(* CODESYS project SIMAI_1.0.0.project

Project tree, tasks and I/O mapping:
  Device : HY-TTC 540, TTControl, order no. n/a, version 1.7.1.0
    application Application
      libraries: Standard, * (System); CAA Can Low Level Extern, * (CAA Technical Workgroup); Util, * (System); SysTypes2 Interfaces, * (System); SysTarget, 3.5.5.0 (System); VisuDialogs, * (System); CAA Memory, 3.5.12.0 (CAA Technical Workgroup); Network, 3.5.7.0 (3S - Smart Software Solutions GmbH); CmpIecTask, * (System); CmpErrors, 3.3.1.40 (System); lib500, 1.7.1.0 (TTControl); lib500_types, 1.7.1.0 (TTControl); lib500_syscom, 1.7.1.0 (TTControl)
      task _NotificationCallback (externalevent, external event NotificationCallback, priority 0) calls _NotificationCB_PRG
      task _ErrorCallback (externalevent, external event ErrorCallback, priority 1) calls _ErrorCB_PRG
      task CommunicationTask (cyclic, interval t#10ms, priority 31, watchdog t#200ms x 1) calls manageGrCommAndEEPROM, CanComunication
      task MainTask (cyclic, interval t#10ms, priority 2, watchdog t#200ms x 1) calls MAIN
      Variable lists/
        global variables GVL
        global variables IO
        global variables fieldbus
        global variables par
        global variables CONST
        global variables ERR
        global variables ui
        global variables CanBusVariables
        global variables EtsdnVar
        global variables EtsOneVar
        global variables system
        global variables RxFlasher
      Program logic/
        program _ErrorCB_PRG [ST]
        program _NotificationCB_PRG [ST]
        Tasks/
          program MAIN [ST]: mainLoop, postrun, shutdown, checkParameters, setupCanbus
          program manageGrCommAndEEPROM [ST]: setVariablesToGrComm, initializeGrCommVariables, initializeEepromStructures
          program CanComunication [ST]: sendVariablesDisplay, receiveVariables, initialize, SendVariablesFromEtsdn, SendVariablesFromEtsOne
        function initializeCanbus [ST]
        program mngCanbusStatus [ST]: checkCanBusStatus
        program UI_PRG [ST]
        TypeApplication/
          program ETSDN_Test_PRG [ST]: endTest, setTestDuration, resetVariablesAndStartTest, mngFailTimer, isRLCurrentFresh
      STRUCTURES/
        data type EEPROM_FLAG
        data type CanHandleStatus
        data type FsmEnum
      Modules/
        IOs/
          Functions/
            program io_module [ST]: instantiateDI, instantiatePWM, instantiatePower, instantiateVOUT, instantiateADC, getInputs, instantiatePWD, initializeIO, instantiateDO, instantiateDIO, instantiatePVG, setOutputs, mngErrors
          Types/
            data type pinPWM
            program initializeIO [ST]: instantiateAnalogInputs, instantiatePVGOutputs, instantiateDigitalOutputs, instantiateVoltageOutputs, instantiatePWDInputs, instantiatePowerStages, instantiatePWMOutputs, instantiateDigitalInputs
            data type type_powerStages
            data type pinADC
            data type type_digitalInputs
            data type pinPVG
            data type type_pwmOutputs
            data type pinPWD
            data type type_voltageOutputs
            data type pinDIO
            data type pwdReadMode
            data type type_digitalOutputs
            data type type_analogInputs
            data type type_pwdInputs
            data type type_pvgOutputs
            data type pin
            data type pinPower
            data type pinVOUT
          global variables sysIO
        COMM/
          Functions/
            program mngCommCan [ST]: mngInit, catchMessages, mngMessage, mngResponse, getsetVarCallback, applyToRamCallback, readAllFromEEPROMCallback, writeToEEPROMCallback, applyToRAM, isVariableValid, initializeVariable
          Types/
            data type grCommVar
            data type grCommAccessRight
            data type grCommVariableStatus
            data type grCommMessageType
            data type grCommEEPROMStatus
          Variable lists/
            global variables grComm
        Canbus/
          Safety interface/
            Tasks/
              program CAN_PRG_SAFE [ST]: exchangeVariables
              program CAN_PRG_UNSAFE [ST]
            Functions/
              program safeSendMessage [ST]
              program safetyCanbusInterface [ST]
              program safeRegisterReceiveMask [ST]
          Variable lists/
            global variables canGVL
            global variables canEVL
          Types/
            data type can
            data type canMessage
            data type canReceiveMask
            data type canBus
          Functions/
            function readMessage [ST]
            program checkReceiveMaskInitialization [ST]
            program registerReceiveMask [ST]
            program sendMessage [ST]
            program initializeCanHandle [ST]
            program checkBusState [ST]
        EEPROM/
          Functions/
            program mngEEPROM [ST]: initEEPROM, mngStep, initializeEepromEntry
          Types/
            Parameters/
              data type HWFW_INFO_TIP
            data type eepromEntry
          Variable lists/
            global variables EEPROM
        Utils/
          program Utils [ST]: decrementUINT, bytesToUInt16, toggle, isNaN, updateValueFiltered, bytesToInt16, decrementUDINT, boolToPWMDutyCycle, linearize, bytesToUReal16, bytesToUDInt32, incrementUINT, getCurrentTaskCycleTime, decrementUINTTimer
        J1939/
          program J1939_PRG [ST]: initReceiveMasks, receiveMessage, parseMessage, sendPGNRequests, mngEngineStatus, redirectToDisplay
          global variables J1939
      visualisation Visualization
    CANs : CANs, TTControl, order no. n/a, version 1.7.1.0
      CAN2 : CAN2, TTControl, order no. n/a, version 1.7.1.0
      CAN3 : CAN3, TTControl, order no. n/a, version 1.7.1.0
      CAN0 : CAN0, TTControl, order no. n/a, version 1.7.1.0
      CAN1 : CAN1, TTControl, order no. n/a, version 1.7.1.0
    System_1 : System, TTControl, order no. n/a, version 1.7.1.0
        unmapped channels: mode, error, mode, error, mode, error, mode, error, mode, error, mode, error, shutdown, error, enable_error_group_0, enable_error_group_1, diag_status, safe_state, error, driver_init_error, UBAT, Terminal_15, WakeUp, Temperature, SSW0, SSW1, SSUP0, SSUP1, SSUP2, status, write, boot_error, trigger_error, Powerstage, SSW0, SSW1, SSUP0, SSUP1, SSUP2, Terminal_15,
          WakeUp, ExtShutOff0, ExtShutOff1
      Timer_Inputs : TIN, TTControl, order no. n/a, version 1.7.1.0
        Pin 147
          <Vuoto>
        Pin 122
          <Vuoto>
        Pin 148
          <Vuoto>
        Pin 146
          <Vuoto>
        Pin 124
          <Vuoto>
        Pin 123
          <Vuoto>
      Analog_Inputs_2Mode_10V : AIN_2Mode_10V, TTControl, order no. n/a, version 1.7.1.0
        Pin 134
          <Vuoto>
        Pin 109
          <Vuoto>
        Pin 132
          <Vuoto>
        Pin 131
          <Vuoto>
        Pin 107
          <Vuoto>
        Pin 110
          <Vuoto>
        Pin 108
          <Vuoto>
        Pin 133
          <Vuoto>
      Analog_Inputs_3Mode : AIN_3Mode, TTControl, order no. n/a, version 1.7.1.0
        Pin 129
          <Vuoto>
        Pin 104
          <Vuoto>
        Pin 130
          <Vuoto>
        Pin 105
          <Vuoto>
        Pin 103
          <Vuoto>
        Pin 127
          <Vuoto>
        Pin 106
          <Vuoto>
        Pin 128
          <Vuoto>
      Digital_Outputs_LS : LSDOUT, TTControl, order no. n/a, version 1.7.1.0
        Pin 239
          <Vuoto>
        Pin 251
          <Vuoto>
        Pin 240
          <Vuoto>
        Pin 252
          <Vuoto>
        Pin 254
          <Vuoto>
        Pin 238
          <Vuoto>
        Pin 253
          <Vuoto>
        Pin 241
          <Vuoto>
      Timer_Inputs_Cur : TIN_Cur, TTControl, order no. n/a, version 1.7.1.0
        Pin 140
          <Vuoto>
        Pin 117
          <Vuoto>
        Pin 116
          <Vuoto>
        Pin 139
          <Vuoto>
        Pin 115
          <Vuoto>
        Pin 141
          <Vuoto>
      Analog_Inputs_2Mode_32V : AIN_2Mode_32V, TTControl, order no. n/a, version 1.7.1.0
        Pin 113
          <Vuoto>
        Pin 137
          <Vuoto>
        Pin 136
          <Vuoto>
        Pin 112
          <Vuoto>
        Pin 138
          <Vuoto>
        Pin 114
          <Vuoto>
        Pin 111
          <Vuoto>
        Pin 135
          <Vuoto>
      PWM_Outputs : PWM, TTControl, order no. n/a, version 1.7.1.0
        Safety_switch_0 : PWM_SSW0, TTControl, order no. n/a, version 1.7.1.0
          Pin 165
            <Vuoto>
          Pin 195
            <Vuoto>
          Pin 162
            <Vuoto>
          Pin 171
            <Vuoto>
          Pin 168
            <Vuoto>
          Pin 186
            <Vuoto>
          Pin 183
            <Vuoto>
          Pin 177
            <Vuoto>
          Pin 180
            <Vuoto>
          Pin 159
            <Vuoto>
          Pin 153
            <Vuoto>
          Pin 189
            <Vuoto>
          Pin 156
            <Vuoto>
          Pin 192
            <Vuoto>
        Safety_switch_1 : PWM_SSW1, TTControl, order no. n/a, version 1.7.1.0
          Pin 157
            <Vuoto>
          Pin 187
            <Vuoto>
          Pin 154
            <Vuoto>
          Pin 160
            <Vuoto>
          Pin 178
            <Vuoto>
          Pin 169
            <Vuoto>
          Pin 166
            <Vuoto>
          Pin 163
            <Vuoto>
          Pin 184
            <Vuoto>
          Pin 181
            <Vuoto>
          Pin 190
            <Vuoto>
          Pin 172
            <Vuoto>
          Pin 193
            <Vuoto>
          Pin 196
            <Vuoto>
      Digital_Outputs_HS : HSDOUT, TTControl, order no. n/a, version 1.7.1.0
        Pin 176
          <Vuoto>
        Pin 149
          <Vuoto>
        Pin 158
          <Vuoto>
        Pin 173
          <Vuoto>
        Pin 152
          <Vuoto>
        Pin 155
          <Vuoto>
        Pin 182
          <Vuoto>
        Pin 179
          <Vuoto>
      Analog_Inputs : AIN, TTControl, order no. n/a, version 1.7.1.0
        Pin 161
          <Vuoto>
        Pin 185
          <Vuoto>
        Pin 188
          <Vuoto>
        Pin 164
          <Vuoto>
        Pin 191
          <Vuoto>
        Pin 167
          <Vuoto>
        Pin 194
          <Vuoto>
        Pin 170
          <Vuoto>
      Digital_Inputs : DIN, TTControl, order no. n/a, version 1.7.1.0
        Pin 101
          <Vuoto>
        Pin 125
          <Vuoto>
        Pin 150
          <Vuoto>
        Pin 174
          <Vuoto>
        Pin 102
          <Vuoto>
        Pin 126
          <Vuoto>
        Pin 151
          <Vuoto>
        Pin 175
          <Vuoto>
  text list GlobalTextList
*)

// Device/Application/STRUCTURES/EEPROM_FLAG
TYPE EEPROM_FLAG : //verificata
STRUCT
	READ: BOOL:= FALSE;
	CHANGED: BOOL:= FALSE;
	WRITE: BOOL:= FALSE;
END_STRUCT
END_TYPE

// Device/Application/Modules/COMM/Types/grCommVar
TYPE grCommVar :
	STRUCT;
		accessRights: grCommAccessRight;
		status: grCommVariableStatus;
		
		pointerToSystemVar: POINTER TO UINT;
		uiLowerValidValue: UINT;
		uiHigherValidValue: UINT;
		uiDefaultValue: UINT;
		
		uiValue: UINT;
	END_STRUCT
END_TYPE

// Device/Application/Modules/COMM/Types/grCommAccessRight
{attribute 'qualified_only'}
{attribute 'strict'}
TYPE grCommAccessRight :
(
	NoAccess := 0,
	ReadOnly := 1,
	ReadWrite := 2
);
END_TYPE

// Device/Application/Modules/COMM/Types/grCommVariableStatus
{attribute 'qualified_only'}
{attribute 'strict'}
TYPE grCommVariableStatus :
(
	Uninitialized:= 0,
	Pristine:= 1,
	ModifiedByRemote:= 2,
	Error:= 3
);
END_TYPE

// Device/Application/Modules/COMM/Types/grCommMessageType
{attribute 'qualified_only'}
{attribute 'strict'}
TYPE grCommMessageType :
(
	ExitCode:= 0,				// Esito di un comando
	
	GetVariable:= 1,			// Get valore di una variabile
	SetVariable:= 2,			// Set valore di una variabile
	HeartRateRequest:= 3,		// Richiesta di heart rate (broadcast)
	LoadFromEEPROM:= 4,			// Leggi parametri da EEPROM
	WriteToEEPROM:= 5,			// Scrivi parametri in RAM sulla EEPROM (rispettando il flag EDIT)
	WriteAllToEEPROM:= 6,		// Scrivi parametri in RAM sulla EEPROM (ignorando il flag EDIT)
	ApplyVariables:= 7,			// Imposta i parametri inviati sulla RAM
	
	ErrorCode:= 255		// Errore
);
END_TYPE

// Device/Application/Modules/IOs/Types/pinPWM
TYPE pinPWM EXTENDS pin :
	STRUCT
		stErrorGetCut: lib500_types.IO_ERRORTYPE;
		wFrequency: WORD:= 100;
		bPolarity: BOOL:= TRUE;
		bDiagMargin: BOOL:= FALSE;
		wFeedbackHighTime: WORD;
		wPeriodFeedback: WORD;
		wCurrent: WORD;
		bCurrentFresh: BOOL;
		wDuty: WORD;
	END_STRUCT
END_TYPE

// Device/Application/Modules/IOs/Types/type_powerStages
TYPE type_powerStages :
STRUCT	
	safetySwitch0: pinPower;	
	safetySwitch1: pinPower;	
	safetySwitch2: pinPower;
	powerStage: pinPower;
	sensorSupply0: pinPower;
	sensorSupply1: pinPower;
	sensorSupply2: pinPower;
END_STRUCT
END_TYPE

// Device/Application/Modules/IOs/Types/pinADC
TYPE pinADC EXTENDS pin :
	STRUCT		
		stADCType: lib500_types.IO_ADC_TYPE;
		stADCRange: lib500_types.IO_ADC_RANGE;
		stADCSensorSupply: lib500_types.IO_SENSOR_SUPPLY;
		dwValue: DWORD;
		bValueFresh: BOOL;
	END_STRUCT
END_TYPE

// Device/Application/Modules/COMM/Types/grCommEEPROMStatus
{attribute 'qualified_only'}
{attribute 'strict'}
TYPE grCommEEPROMStatus :
(
	Idle:= 0,
	BeginRead:= 1,
	Reading:= 2,
	BeginWrite:= 3,
	Writing
);
END_TYPE

// Device/Application/Modules/IOs/Types/type_digitalInputs
TYPE type_digitalInputs :
STRUCT	
	fuelReserve_p127: pinDIO;

	xSensorUltra_OSSID11_p115: pinDIO; 
	xSensorUltra_OUT1_p116: pinDIO; 
	
	xSensorUltra_OSSID21_p139: pinDIO; 
	xSensorUltra_OUT2_p140: pinDIO; 	
	
	xRadioAutecFwd_p117: pinDIO; 	
	
	xStraightWheels_p141: pinDIO; 
END_STRUCT
END_TYPE

// Device/Application/Modules/IOs/Types/pinPVG
TYPE pinPVG EXTENDS pin :
	STRUCT
		stGetVoltageError: lib500_types.IO_ERRORTYPE;
		wValue: WORD := 5000;
		uiReadVoltage: UINT := 0;
		bVoltageFresh: BOOL := FALSE;
	END_STRUCT
END_TYPE

// Device/Application/Modules/Canbus/Types/can
TYPE can :
	STRUCT
			
		bInitialized: BOOL:= FALSE;	
		usiChannel: USINT:= 0;
		uiBaudrateKbps: UINT:= 0;
	
		driver: CL2.CAA.HANDLE;
		initializeError: CL2.ERROR;
		transmitError: CL2.ERROR;
		busStatus: CL2.BUSSTATE;
		
		receiveMessageHandle: CL2.CAA.HANDLE := CL2.CAA.gc_hINVALID;
		pointerToData: POINTER TO CL2.CL2I.DATA;
		messageLeft : CL2.CAA.COUNT;
		
		uiMessageCount: INT:=0;
		byaReceiveBuffer: ARRAY [0..7] OF BYTE;				
		byaTransmitBuffer: ARRAY [0..7] OF BYTE;						
		
	END_STRUCT
END_TYPE

// Device/Application/Modules/IOs/Types/type_pwmOutputs
TYPE type_pwmOutputs :
STRUCT
	turtleBtnBacklight_p168: pinPWM;
END_STRUCT
END_TYPE

// Device/Application/Modules/Canbus/Types/canMessage
TYPE canMessage :
	STRUCT
		udiId: UDINT:= 0;
		bExtended: BOOL:= FALSE;
		byLength: BYTE:= 8;
		byaData: ARRAY [0..7] OF BYTE;
	END_STRUCT
END_TYPE

// Device/Application/Modules/Canbus/Types/canReceiveMask
TYPE canReceiveMask :
	STRUCT
		bActive: BOOL:= FALSE;
		bInitialized: BOOL:= FALSE;
		udiId: UDINT:= 0;
		stCAAMask: CL2.CAA.HANDLE:= CL2.CAA.gc_hINVALID;	
		stMessagesLeft: CL2.CAA.COUNT;	
		udiCobIdMask: UDINT:= 16#1FFFFFFF;
	END_STRUCT
END_TYPE

// Device/Application/Modules/Canbus/Types/canBus
TYPE canBus :
	STRUCT
		bActive: BOOL:= FALSE;
		stChannel: can;
		staReceiveMasks: ARRAY[0..canGVL.iReceiveMaskCount-1] OF canReceiveMask;
		stTransmitBuffer: ARRAY[0..canGVL.iTransmitBufferSize-1] OF canMessage;
	END_STRUCT
END_TYPE

// Device/Application/Modules/IOs/Types/pinPWD
TYPE pinPWD EXTENDS pin :
	STRUCT
		stGetVoltageError: lib500_types.IO_ERRORTYPE;
		stIncSetError: lib500_types.IO_ERRORTYPE;
		pwdMode: lib500_types.IO_PWD_INC_MODE;
		wCountInit: WORD:= 32767;
		wCount: WORD;
		wCountZero: WORD;
		uiVoltage: UINT;
		bChannelA: BOOL;
		bChannelB: BOOL;
		readMode: pwdReadMode;
		pulseSamples: lib500_types.IO_PWD_PULSE_SAMPLES;
		dwFrequencyHz: DWORD;
		dwPulseWidth: DWORD;
		pulseMode: lib500_types.IO_PWD_PULSE_MODE;
		freqMode: lib500_types.IO_PWD_FREQ_MODE;
		byCaptureCount: BYTE;
		bVoltageFresh: BOOL;
		bSetIncrementCount: BOOL:= FALSE;
	END_STRUCT
END_TYPE

// Device/Application/Modules/IOs/Types/type_voltageOutputs
TYPE type_voltageOutputs :
STRUCT
	etsAI10V_p185: pinVOUT;
	etsAI5V_p161: pinVOUT;
	// dummy: pinVOUT;
END_STRUCT
END_TYPE

// Device/Application/STRUCTURES/CanHandleStatus
TYPE CanHandleStatus :
	STRUCT
		uidFreeMessagesInPoll: UDINT:= 0;
		uidMessagesInElabQueue: UDINT:= 0;
	END_STRUCT
END_TYPE

// Device/Application/Modules/IOs/Types/pinDIO
TYPE pinDIO EXTENDS pin :
	STRUCT
		bValue: BOOL:= FALSE;
		wCurrent: WORD;
		bCurrentFresh: BOOL;
		stErrorGetCut: lib500_types.IO_ERRORTYPE;
	END_STRUCT
END_TYPE

// Device/Application/Modules/IOs/Types/pwdReadMode
{attribute 'qualified_only'}
{attribute 'strict'}
TYPE pwdReadMode :
(
	incremental := 0,
	complex
);
END_TYPE

// Device/Application/Modules/IOs/Types/type_digitalOutputs
TYPE type_digitalOutputs :
STRUCT				 
	etsPower_p177: pinDIO;
	etsIP1_p188: pinDIO;
	etsIP2_p164: pinDIO;
	
	etsRele_p180: pinDIO;
	etsRele_p183: pinDIO;
	etsRele_p186: pinDIO;
	
	
	etsIN1_p251: pinDIO;
	etsIN2_p238: pinDIO;
	
	
	etsonePower_p153: pinDIO;
	
	etsoneRele_p156: pinDIO;
	etsoneRele_p159: pinDIO;
	
	etsoneIP3_p194: pinDIO;
END_STRUCT
END_TYPE

// Device/Application/Modules/IOs/Types/type_analogInputs
TYPE type_analogInputs :
STRUCT
	ecuK15_p207: pinADC;
	
	ets5V_p131: pinADC;
	etsone5V_107: pinADC;
END_STRUCT
END_TYPE

// Device/Application/Modules/IOs/Types/type_pwdInputs
TYPE type_pwdInputs :
STRUCT
	transmissionShaftSensor5000_p175: pinPWD;
	transmissionShaftSensor7500_p151: pinPWD;
END_STRUCT
END_TYPE

// Device/Application/Modules/IOs/Types/type_pvgOutputs
TYPE type_pvgOutputs :
STRUCT
	//_p161: pinPWD;
END_STRUCT
END_TYPE

// Device/Application/Modules/IOs/Types/pin
TYPE pin :
	STRUCT
		bInitialized: BOOL:= FALSE;
		stInitError: lib500_types.IO_ERRORTYPE;
		stError: lib500_types.IO_ERRORTYPE;
		byChannel: BYTE;
		byPullType: BYTE;
		byMinTTCModel: BYTE:= 0;
		byResetCount: BYTE:= 0;
	END_STRUCT
END_TYPE

// Device/Application/Modules/IOs/Types/pinPower
TYPE pinPower EXTENDS pin :
	STRUCT
		mode: lib500_types.IO_POWER_STATE;
	END_STRUCT
END_TYPE

// Device/Application/Modules/EEPROM/Types/eepromEntry
TYPE eepromEntry :
	STRUCT
		wAddress: WORD;
		pData: POINTER TO BYTE;
		wSize: WORD;
	END_STRUCT
END_TYPE

// Device/Application/Modules/EEPROM/Types/Parameters/HWFW_INFO_TIP
TYPE HWFW_INFO_TIP :
	STRUCT		
		PASSWORD_LEVEL_0: UINT:= 0;
		PASSWORD_LEVEL_1: UINT:= 1234;		
	END_STRUCT
END_TYPE

// Device/Application/Modules/IOs/Types/pinVOUT
TYPE pinVOUT EXTENDS pin :
	STRUCT
		wOutputVoltageMv: WORD:= 0;
	END_STRUCT
END_TYPE

// Device/Application/STRUCTURES/FsmEnum
{attribute 'qualified_only'}
{attribute 'strict'}
TYPE FsmEnum :
(
	FSM_WAIT00 := 0,
	FSM_STOP,
	FSM_RUN
);
END_TYPE

// Device/Application/Modules/COMM/Variable lists/grComm
{attribute 'qualified_only'}

(* User code configurable settings *)
VAR_GLOBAL CONSTANT
	uiProtocolMessageID : UINT:=16#7F7;
	uiProtocolVirtualNode : UINT:=16#3;	
	uiVariablesMaxIndex: UINT:= 100;    // Reduce this value if you have low memory issues
END_VAR



(* User code accessible status variables *)
VAR_GLOBAL  			
	bCommunicationActive: BOOL:=FALSE;			// Indicates that a communication is running
	bTriggerReadFromEEPROM: BOOL:= TRUE;		// If active user code should read variables from EEPROM and store their value in grComm.staVariables
	bTriggerApplyToRAM: BOOL:= FALSE;			// If active user code should set its system values from grComm.staVariables
	bTriggerWriteToEEPROM: BOOL:= FALSE;		// If active user code should write to EEPROM only the modified variable's values from grComm.staVariables
	bTriggerWriteAllToEEPROM: BOOL:= FALSE;		// If active user code should write to EEPROM all the variable's values from grComm.staVariables
END_VAR


(* Internal logic variables *)
VAR_GLOBAL
	staVariables: ARRAY[1..uiVariablesMaxIndex] OF grCommVar;	
END_VAR

(* Internal logic defines *)
VAR_GLOBAL CONSTANT	
	COMM_TIMER_RLD: UINT:= 1000;
	LIB_VERSION_CODE: BYTE:= 0;		
	
	// Exit code viene messo nel campo ADDRESS se TYPE == EXIT_CODE
	EXIT_CODE_ERROR: UINT:= 0;
	EXIT_CODE_OK: UINT:= 1;

END_VAR

// Device/Application/Variable lists/GVL
{attribute 'qualified_only'}
VAR_GLOBAL
	MODELLO_CENTRALINA: BYTE;
	fwVersion: ARRAY[0..2] OF BYTE:= [1, 0, 0];  // versione di cenrtralina 3.0.0
	
	xAllowSystemShutdown: BOOL;
END_VAR

// Device/Application/Variable lists/IO
{attribute 'qualified_only'}
VAR_GLOBAL
	xECUK15: BOOL;

	xSensorUltra_10 : UINT;
END_VAR

// Device/Application/Modules/Canbus/Variable lists/canGVL
{attribute 'qualified_only'}

VAR_GLOBAL CONSTANT	
	iBusCount: INT:= 10;
	iTransmitBufferSize: INT:= 50;
	iReceiveMaskCount: INT:= 50;
END_VAR

VAR_GLOBAL
	busses: ARRAY[0..iBusCount-1] OF canBus;
END_VAR

// Device/Application/Variable lists/fieldbus
{attribute 'qualified_only'}
VAR_GLOBAL CONSTANT
	iCanbusCount: INT:= 4;
	uiaCanBaudrates: ARRAY[0..9] OF UINT:= [500, 250, 500, 500, 1000, 0, 0, 0, 0, 0];
END_VAR

VAR_GLOBAL
	can: ARRAY [0..9] OF canBus;
	
	bCanbusInitialized: BOOL:= FALSE;
END_VAR

// Device/Application/Variable lists/par
{attribute 'qualified_only'}
VAR_GLOBAL
	stHwFwInfo: HWFW_INFO_TIP;
END_VAR

// Device/Application/Variable lists/CONST
{attribute 'qualified_only'}
VAR_GLOBAL	
	CANBUS_MAX_READS_PER_CYCLE: BYTE:= 10;
	CANBUS_MIN_FREE_POLL: BYTE:= 30;
	CANBUS_MAX_RX_QUEUE: BYTE:= 15;
END_VAR

// Device/Application/Modules/IOs/sysIO
{attribute 'qualified_only'}
VAR_GLOBAL
	bIOInstantiated: BOOL:= FALSE;
	bIOInitialized: BOOL:= FALSE;

	digitalInput: type_digitalInputs;
	analogInput: type_analogInputs;
	pwdInput: type_pwdInputs;
	pvgOutput: type_pvgOutputs;
	
	digitalOutput: type_digitalOutputs;
	powerStage: type_powerStages;
	pwmOutput: type_pwmOutputs;
	voltageOutput: type_voltageOutputs;
END_VAR

// Device/Application/Modules/Canbus/Variable lists/canEVL
(* THIS EVL IS AUTOGENERATED. DO NOT MODIFY THESE ATTRIBUTES. *)
{attribute 'location' := '16#800' }
{attribute 'linkalways'}
{attribute 'qualified_only'}
VAR_GLOBAL	
	bHasChanges: BOOL:= FALSE;
	bChannelsHasChanges: BOOL:= FALSE;
	bTransmitBuffersHasChanges: BOOL:= FALSE;
	bMasksHasChanges: BOOL:= FALSE;
	busses: ARRAY[0..canGVL.iBusCount-1] OF canBus;
END_VAR

// Device/Application/Modules/EEPROM/Variable lists/EEPROM
{attribute 'qualified_only'}

(* User code accessible status indicators *)
VAR_GLOBAL
	bTriggerReadAll: BOOL:= FALSE;
	
	bEEPROMInitialized: BOOL := FALSE;
	bReadFromEEPROM: BOOL := TRUE;
	bWriteAllToEEPROM: BOOL:= FALSE;
END_VAR


(* Internal logic *)
VAR_GLOBAL CONSTANT	
	iEepromEntriesCount: INT:= 160;
END_VAR
VAR_GLOBAL	
	staAllEntries: ARRAY[0..iEepromEntriesCount-1] OF eepromEntry; // On TTC-500 series EEPROM is 64KB. Each structure has 400 byte of space reserved
END_VAR

// Device/Application/Variable lists/ERR
{attribute 'qualified_only'}
VAR_GLOBAL
	xInputPins: BOOL;
	xOutputPins: BOOL;
	xInitializePins: BOOL;
	xCanbusHeavy: BOOL;
END_VAR

// Device/Application/Variable lists/ui
{attribute 'qualified_only'}
VAR_GLOBAL
	xBlinker_100ms: BOOL;
	xBlinker_500ms: BOOL;
END_VAR

// Device/Application/Modules/J1939/J1939
{attribute 'qualified_only'}
VAR_GLOBAL
	byECUNodeId: BYTE:= 16#10;
	xEngineOnline: BOOL:= FALSE;
	xSendPGNRequest: BOOL:= FALSE;
	xRedirectMessages: BOOL:= FALSE;
	
	// valori in arrivo dal bus
	iTorquePercent: INT;
	uiEngineSpeedRpm: UINT;
	uiMinutesRunWhileMILAct: UINT;
	lrEngineTotalFuelUsedLiters: LREAL;
	rEngineFuelRateLph: REAL;
	byBarometricPressureKPa: BYTE;
	iAmbientAirTemperatureDegC: INT;
	iEngineIntakeAirTemperatureDegC: INT;
	uiOilPressureKPa: UINT;
	byCoolantLevelPerc: BYTE;
	iEngineCoolantTempDegC: INT;
	iEngineFuelTempDegC: INT;
	iAftertreatmentDPFIntakeGasTempDegC: INT;
	rBatteryPotentialV: REAL;
	byEngineStartEnable: BYTE;
	rEngineTotalIdleHours: REAL;
	byAftertreatmentEngineSpeedIncreaseRequest: BYTE;
	byEngineWaitToStartLamp: BYTE;
	byEngineIdleShutdownStatus: BYTE;
	byEngineIdleShutdownAlert: BYTE;
	byServiceComponentId1: BYTE;
	byServiceComponentId2: BYTE;
	byServiceComponentId3: BYTE;
	iServiceDelayHours: INT;
	rEngineTotalOperationHours: REAL;
	byDPFFilterLamp: BYTE;
	byAftertreatmentDPFActiveRegeneration: BYTE;
	byAftertreatmentDPFFilterStatus: BYTE;
	byDPFActiveRegenerationInhibitedDueSwitch: BYTE;
	byDPFActiveRegenerationInhibitedDueTmpSysLock: BYTE;
	byDPFActiveRegenerationInhibitedDuePermSysLock: BYTE;
	
	
	byWarningIndicator: BYTE;	
	byWarningIndicatorFlash: BYTE;
	byShutdownIndicator: BYTE;
	byEngineProtectIndicator: BYTE;
	byEngineProtectIndicatorFlash: BYTE;
	byEmissionSystemMalfunctionIndicator: BYTE;
	byEmissionSystemMalfunctionIndicatorFlash: BYTE;	
	
	
	// trouble codes
	DM1_SPN: ULINT;
	DM1_FMI: UINT;
	DM1_OC: UINT;
	
	
	// valori calcolati
	xEngineRunning: BOOL;
	xEngineDPFRegenRequest: BOOL;
	xEngineDPFRegenActive: BOOL;
	xLowOilPressure: BOOL;
	xEngineLamp: BOOL;
	xEngineLampRed: BOOL;
	byRegenerationStatus: BYTE;
	
	
END_VAR

// Device/Application/Variable lists/CanBusVariables
{attribute 'qualified_only'}
VAR_GLOBAL
	(* variabili lette su CanBus  *) 
    sSteeringAngle: SINT;
	
	
	
	(* derivate da variabili lette su CanBus  *) 
	xWheelAlignment: BOOL;
END_VAR

// Device/Application/Variable lists/EtsdnVar
{attribute 'qualified_only'}
VAR_GLOBAL
		
	cmdTest : BYTE;  // comando del test che arriva dal Flasher

	xOnline: BOOL;  // stato online del CAN ( comunicazione attiva )
	
	(* Inviati da pc a Plc *)
	xRL1: BOOL;  // richiesta attivazione relè 1 (da plc a Etsdn )
	xRL2: BOOL;  // richiesta attivazione relè 2 (da plc a Etsdn )
	xRL3: BOOL;  // richiesta attivazione relè 3 (da plc a Etsdn )
	xPwrSupplyRL1: BOOL;   // richiesta alimentazione relè 1 (da plc a Etsdn )
	xPwrSupplyRL2: BOOL;   // richiesta alimentazione relè 2 (da plc a Etsdn )
	xPwrSupplyRL3: BOOL;   // richiesta alimentazione relè 3 (da plc a Etsdn )
	
	xPwrSupplyIP1: BOOL;   // richiesta alimentazione Ingresso Positivo 1 (da plc a Etsdn )
	xPwrSupplyIP2: BOOL;   // richiesta alimentazione Ingresso Positivo 1  (da plc a Etsdn )
	xPwrSupplyIN1: BOOL;   // richiesta alimentazione Ingresso Negativo 1 (da plc a Etsdn )
	xPwrSupplyIN2: BOOL;   // richiesta alimentazione Ingresso Negativo 1  (da plc a Etsdn )
	xCycle10V: BOOL; 		//richiesta ciclo dei 10 volt (da plc a Etsdn )
	xCycle5V: BOOL; 		//richiesta ciclo dei 5 volt (da plc a Etsdn )
	(* Ricevuti da Etsdn *)
	xIP1: BOOL;   // stato dell'ingresso digitale positivo IP1 (da Etsdn a plc ) associato a etsIP1_p188.
	xIP2: BOOL;   // stato dell'ingresso digitale positivo IP2 (da Etsdn a plc ) associato a etsIP2_p164
	xIN1: BOOL;   // stato dell'ingresso digitale negativo IN1 (da Etsdn a plc ) associato a etsIN1_p251
	xIN2: BOOL;   // stato dell'ingresso digitale negativo IN2 (da Etsdn a plc ) associato a etsIN2_p238
	
	rAI: REAL;    // 5V
	rIP3: REAL;   // 10V
	
	rX: REAL;
	rY: REAL;
	rZ: REAL;
	
	rSupplyVoltage: REAL;
	
	(* metto i messaggi ricevuti in queste strutture per poi rimandarli al Flasher  *)
	msgRx_01 :ARRAY[0..7] OF BYTE;
	msgRx_02 :ARRAY[0..7] OF BYTE;
	msgRx_03 :ARRAY[0..7] OF BYTE;
	
	
	 
	
END_VAR

// Device/Application/Variable lists/EtsOneVar
{attribute 'qualified_only'}
VAR_GLOBAL
	// Ricevuti da Flasher
	cmdTest: BYTE;
	
	// Inviati al Flasher

	
	
	xOneRL1: BOOL; 
	xOneRL2: BOOL; 
	rPwrSupplyOneRL1: WORD;
	rPwrSupplyOneRL2: WORD;
	
	xOneIP1: BOOL;
	xOneIP2: BOOL;
	xOneIP3: BOOL;
	xCycleOneIP4: BOOL;
 
	xOne5V: BOOL;
	dwOne5V: DWORD;
END_VAR

// Device/Application/Variable lists/system
{attribute 'qualified_only'}
VAR_GLOBAL CONSTANT	
	FWV_PRIMARIA: BYTE:=0;
	FWV_SECONDARIA: BYTE:=0;
	FWV_BUGFIX: BYTE:=0;	
END_VAR

VAR_GLOBAL	
	xFirstCycle: BOOL:= TRUE;
	
	fwVMergedPrimarySecondary: UINT:= (FWV_PRIMARIA * 256) OR FWV_SECONDARIA;
	fwVMergedRevisionBugfix: UINT:= FWV_BUGFIX;
	bHasAlarms: BOOL:= FALSE;	
	
	matricolaL: UINT:= 0;
	matricolaH: UINT:= 0;
	
	bParametersReady: BOOL:= FALSE;	
	systemAlarms: UINT:= 0;
	
	xHazardStatus: BOOL:= FALSE;
	xParkingBrakeActive: BOOL:= FALSE;
	xInchingModeActive: BOOL:= FALSE;
	
	byActiveGear: BYTE:= 0;
	byDirection: BYTE:= 0;
	byFuelPercent: BYTE;
	
	xSeatStatus: BOOL;
	rFuelLevelFiltered: REAL;
	udiInchingAlertTimerMs: UDINT;
	
	rSpeedKmph: REAL;
	xIncorrectStart: BOOL;
	
		
	xTestRunning: BOOL;
	xTestResultValid: BOOL;
	xTestResult: BOOL;
	xCanTestResult: BOOL;
	xDigitalInTestResult: BOOL;
	xAnalogInTestResult: BOOL;
	xPowerTestResult: BOOL;
	x5VOutTestResult: BOOL;
	xAccelerometerTestResult: BOOL;
	xReleTestResult: BOOL;
	
	iAccTestStep: INT:= -1;
	byTestPercentage: BYTE;
	
END_VAR

// Device/Application/Variable lists/RxFlasher
{attribute 'qualified_only'}
VAR_GLOBAL
	systemUnderTest : BYTE := 0;  // 0=nessun0 1=Etsdn	2=Mdt
END_VAR

// Device/Application/Program logic/_NotificationCB_PRG
PROGRAM _NotificationCB_PRG
VAR
	diag_state : lib500_types.DIAG_STATETYPE := lib500_types.DIAG_STATETYPE.DIAG_STATE_DISABLED;
	watchdog_state : lib500_types.DIAG_WD_STATETYPE := lib500_types.DIAG_WD_STATETYPE.DIAG_WD_STATE_UNKNOWN;
	error : lib500_types.DIAG_ERRORCODE := (error_code := lib500_types.DIAG_ERRORTYPE.DIAG_E_NOERROR, 
                                            device_num := lib500_types.DIAG_DEVICETYPE.DIAG_DEV_NONE,
                                            faulty_value := 0);
	return_code : lib500_types.IO_ERRORTYPE := lib500_types.IO_ERRORTYPE.IO_E_UNKNOWN;
	
	call_count : UDINT := 0;
END_VAR

(* get the reason for the notification callback *)
return_code := lib500.DIAG_CDS_GetNotificationReason(ADR(diag_state), 
                                                     ADR(watchdog_state),
                                                     ADR(error));

(* custom handler code can be placed here *)

(* increment call count *)
call_count := call_count + 1;

END_PROGRAM

// Device/Application/Program logic/_ErrorCB_PRG
PROGRAM _ErrorCB_PRG
VAR
	diag_state : lib500_types.DIAG_STATETYPE := lib500_types.DIAG_STATETYPE.DIAG_STATE_DISABLED;
	watchdog_state : lib500_types.DIAG_WD_STATETYPE := lib500_types.DIAG_WD_STATETYPE.DIAG_WD_STATE_UNKNOWN;
	error : lib500_types.DIAG_ERRORCODE := (error_code := lib500_types.DIAG_ERRORTYPE.DIAG_E_NOERROR, 
                                            device_num := lib500_types.DIAG_DEVICETYPE.DIAG_DEV_NONE,
                                            faulty_value := 0);
	return_code : lib500_types.IO_ERRORTYPE := lib500_types.IO_ERRORTYPE.IO_E_UNKNOWN;
	
	reaction : lib500_types.DIAG_REACTION := lib500_types.DIAG_REACTION.DIAG_ERR_SAFESTATE;
	
	call_count : UDINT := 0;
END_VAR

(* get the reason for the error callback *)
return_code := lib500.DIAG_CDS_GetErrorReason(ADR(diag_state), 
                                              ADR(watchdog_state),
                                              ADR(error));

(* custom handler code can be placed here *)

(* the choices for the reactions are:
   -> lib500_types.DIAG_REACTION.DIAG_ERR_NOACTION
   -> lib500_types.DIAG_REACTION.DIAG_ERR_SAFESTATE
   -> lib500_types.DIAG_REACTION.DIAG_ERR_DISABLE_SSW0
   -> lib500_types.DIAG_REACTION.DIAG_ERR_DISABLE_SSW1
   -> lib500_types.DIAG_REACTION.DIAG_ERR_DISABLE_SSW2
   -> lib500_types.DIAG_REACTION.DIAG_ERR_DISABLE_HS00
   -> lib500_types.DIAG_REACTION.DIAG_ERR_DISABLE_HS01
   -> lib500_types.DIAG_REACTION.DIAG_ERR_DISABLE_HS02
   -> lib500_types.DIAG_REACTION.DIAG_ERR_DISABLE_HS03
   -> lib500_types.DIAG_REACTION.DIAG_ERR_DISABLE_HS04
   -> lib500_types.DIAG_REACTION.DIAG_ERR_DISABLE_HS05
   -> lib500_types.DIAG_REACTION.DIAG_ERR_DISABLE_HS06
   -> lib500_types.DIAG_REACTION.DIAG_ERR_DISABLE_HS07
   
   it's also possible to combine (binary-or) reactions, like:
   -> lib500_types.DIAG_REACTION.DIAG_ERR_DISABLE_SSW0 OR 
      lib500_types.DIAG_REACTION.DIAG_ERR_DISABLE_SSW1
*)

(* pass the error reaction to the DIAG system *)
lib500.DIAG_CDS_SetErrorReaction(reaction);

(* increment call count *)
call_count := call_count + 1;

END_PROGRAM

// Device/Application/Program logic/Tasks/manageGrCommAndEEPROM
PROGRAM manageGrCommAndEEPROM
VAR
	bGrCommInitialized: BOOL:= FALSE;
	bEepromStructuresInitialized: BOOL:= FALSE;
	uiDummy: UINT:= 0;
END_VAR

(* 
*  You must respect this priorities to allow grComm to 
*  always give a consistent value to the variables 
*)
IF NOT bEepromStructuresInitialized THEN
	bEepromStructuresInitialized:= initializeEepromStructures();
	
ELSIF NOT bGrCommInitialized THEN
	bGrCommInitialized:= initializeGrCommVariables();
	
ELSIF grcomm.bTriggerReadFromEEPROM THEN
	EEPROM.bReadFromEEPROM:= TRUE;
	grcomm.bTriggerReadFromEEPROM:= FALSE;

ELSIF EEPROM.bReadFromEEPROM THEN
	mngEEPROM();
	bGrCommInitialized:= EEPROM.bReadFromEEPROM; 							// when reading has ended, triggers initialization 
	IF NOT EEPROM.bReadFromEEPROM THEN system.bParametersReady:= TRUE; END_IF	// when reading has ended, activate parameters ready flag

ELSIF grcomm.bTriggerApplyToRAM THEN
	mngCommCan.applyToRAM();
	grcomm.bTriggerApplyToRAM:= FALSE;

ELSIF (grcomm.bTriggerWriteToEEPROM OR grcomm.bTriggerWriteAllToEEPROM) THEN
	EEPROM.bWriteAllToEEPROM:= TRUE;
	grcomm.bTriggerWriteToEEPROM:= FALSE;
	grcomm.bTriggerWriteAllToEEPROM:= FALSE;

ELSIF EEPROM.bWriteAllToEEPROM THEN
	mngEEPROM();
	EEPROM.bReadFromEEPROM:= EEPROM.bReadFromEEPROM; // when reading has ended, triggers read from eeprom
	
ELSE
	setVariablesToGrComm();
	mngCommCan(stCanbus:= fieldbus.can[1]);
END_IF

METHOD PRIVATE setVariablesToGrComm
VAR
	uiVarIterator: UINT;
END_VAR
FOR uiVarIterator:= 1 TO grComm.uiVariablesMaxIndex BY 1 DO
	IF mngCommCan.isVariableValid(grComm.staVariables[uiVarIterator]) AND (grComm.staVariables[uiVarIterator].status <> grCommVariableStatus.ModifiedByRemote) THEN
		grComm.staVariables[uiVarIterator].uiValue:= grComm.staVariables[uiVarIterator].pointerToSystemVar^;
	END_IF
END_FOR
END_METHOD

METHOD PRIVATE initializeGrCommVariables : BOOL
VAR_INPUT
END_VAR
(* user code should setup the desired addresses like this 
*      grComm.staVariables[ <NETWORK_ADDR> ]:= mngCommCan.initializeVariable(
*										pointerToSystemVar:= ADR( <SYS_VARIABLE> ),
*										accessRights:= grCommAccessRight.ReadOnly,
*										uiDefaultValue:= x,
*										uiLowerValidValue:= y,
*										uiHigherValidValue:= z
*									);
*  use the variable address as the array index.
*  You can make the code more readable passing the arguments without naming it
*)		
		
grComm.staVariables[2]:= 		mngCommCan.initializeVariable(ADR(uiDummy),		grCommAccessRight.ReadOnly, 1, 0, 16#FFFF);
grComm.staVariables[3]:= 		mngCommCan.initializeVariable(ADR(uiDummy),		grCommAccessRight.ReadOnly, 1, 0, 16#FFFF);
grComm.staVariables[4]:= 		mngCommCan.initializeVariable(ADR(uiDummy),		grCommAccessRight.ReadOnly, 1, 0, 16#FFFF);


grComm.staVariables[9]:= 		mngCommCan.initializeVariable(ADR(system.systemAlarms),						grCommAccessRight.ReadWrite, 0, 0, 16#FFFF);

grComm.staVariables[16#0A]:=	mngCommCan.initializeVariable(ADR(par.stHwFwInfo.PASSWORD_LEVEL_0),		grCommAccessRight.ReadWrite, 0, 	0, 16#FFFF);
grComm.staVariables[16#0B]:=	mngCommCan.initializeVariable(ADR(par.stHwFwInfo.PASSWORD_LEVEL_1),		grCommAccessRight.ReadWrite, 1234, 	0, 16#FFFF);


initializeGrCommVariables:= TRUE;
END_METHOD

METHOD PRIVATE initializeEepromStructures : BOOL
VAR_INPUT
END_VAR
mngEEPROM.initializeEepromEntry(wAddress:= 16#0000, pData:= ADR(par.stHwFwInfo), wSize:= SIZEOF(par.stHwFwInfo));

initializeEepromStructures:= TRUE;
END_METHOD

END_PROGRAM

// Device/Application/Modules/EEPROM/Functions/mngEEPROM
PROGRAM mngEEPROM
VAR	
	eepromErrorCode : lib500_types.IO_ERRORTYPE := lib500_types.IO_ERRORTYPE.IO_E_OK;
	eepromStatus : lib500_types.IO_ERRORTYPE := lib500_types.IO_ERRORTYPE.IO_E_OK;
	eepromLoopStep : INT:=0;
	
	eepromBusy: BOOL:= FALSE;
	iEntryCursor: INT:= 0;
END_VAR

IF NOT EEPROM.bEEPROMInitialized THEN
	initEEPROM();

ELSIF (NOT EEPROM.bReadFromEEPROM) AND (NOT EEPROM.bWriteAllToEEPROM) THEN
	RETURN;
	
ELSE		
	
	mngStep(uiAddress:= EEPROM.staAllEntries[eepromLoopStep].wAddress, 
			bRead:= EEPROM.bReadFromEEPROM, 
			pData:= EEPROM.staAllEntries[eepromLoopStep].pData, 
			wLength:= EEPROM.staAllEntries[eepromLoopStep].wSize);

	(* eepromLoopStep is incremented by mngStep function *)			
	IF (EEPROM.staAllEntries[eepromLoopStep].pData = 0) THEN				
		EEPROM.bReadFromEEPROM:= FALSE;
		EEPROM.bWriteAllToEEPROM:= FALSE;
		eepromLoopStep:= 0;	
	END_IF
	
END_IF

ACTION initEEPROM:
eepromErrorCode := lib500.IO_EEPROM_Init();		
eepromStatus := lib500.IO_EEPROM_GetStatus();
EEPROM.bEEPROMInitialized:= (eepromStatus = lib500_types.IO_ERRORTYPE.IO_E_OK);
END_ACTION

METHOD mngStep
VAR_INPUT
	bRead: BOOL;
	uiAddress: UINT;
	pData: POINTER TO BYTE;
	wLength: WORD;
END_VAR
IF NOT eepromBusy THEN	
	eepromErrorCode := lib500.IO_EEPROM_GetStatus();
	IF (eepromErrorCode = lib500_types.IO_ERRORTYPE.IO_E_OK) THEN
		eepromBusy:= TRUE;
		IF bRead THEN
			eepromErrorCode := lib500.IO_EEPROM_Read(offset:= uiAddress, length:= wLength, data:= pData);
		ELSE
			eepromErrorCode := lib500.IO_EEPROM_Write(offset:= uiAddress, length:= wLength, data:= pData);
		END_IF
	END_IF
	
ELSIF eepromBusy AND eepromStatus = lib500_types.IO_ERRORTYPE.IO_E_OK THEN
	eepromBusy:= FALSE;
	eepromLoopStep:= eepromLoopStep+1;
	
END_IF
END_METHOD

METHOD PUBLIC initializeEepromEntry
VAR_INPUT
	wAddress: WORD;
	pData: POINTER TO BYTE;
	wSize: WORD;
END_VAR
EEPROM.staAllEntries[iEntryCursor].wAddress:= wAddress;
EEPROM.staAllEntries[iEntryCursor].pData:= pData;
EEPROM.staAllEntries[iEntryCursor].wSize:= wSize;

iEntryCursor:= iEntryCursor+1;
IF (iEntryCursor >= EEPROM.iEepromEntriesCount) THEN
	iEntryCursor:= 0;
END_IF
END_METHOD

END_PROGRAM

// Device/Application/Modules/COMM/Functions/mngCommCan
// This PRG contains non safety-related code.
// The following attribute is autogenerated. Do not remove.
{attribute 'location':='16#800'}
PROGRAM mngCommCan

VAR CONSTANT 
	MAX_LOOP: BYTE:=20;
END_VAR

VAR_INPUT	
	stCanbus: canBus;
END_VAR
VAR	
	init : BOOL := FALSE;
	stReceiveMaks: canReceiveMask;
	
	MISSED_COUNTER: UINT:= 0;
	LOOP_COUNTER: BYTE;
	COMM_TIMER: UINT :=0;
	eError : CL2.ERROR;
	SEND_Error : CL2.ERROR;
	BUSSTATE:CL2.BUSSTATE;

	hCAN_RX : CL2.CAA.HANDLE := CL2.CAA.gc_hINVALID;
		
	hRxMsg : CL2.CAA.HANDLE := CL2.CAA.gc_hINVALID;
	pRxData : POINTER TO CL2.CL2I.DATA;
	ctMsgLeft : CL2.CAA.COUNT;
	
	CAN_RX_COUNT: INT:=0;
	CAN_RX_BUFFER	: ARRAY [0..7] OF BYTE;		
	CAN_TX_BUFFER	: ARRAY [0..7] OF BYTE;		

	CMD_ADDR: UINT:=0;
	CMD_PROG: UINT:=0;
	CMD_DATA: UINT:=0;
	CMD_DNODE: UINT:=0;
	CMD_SNODE: UINT:=0;
	CMD_TYPE: BYTE:=0;
	CMD_FREE: BYTE:=0;
		
	TX_COMM: BOOL:=FALSE;
	
	RSP_ADDR: UINT:=0;
	RSP_PROG: UINT:=0;
	RSP_DATA: UINT:=0;
	RSP_DNODE: UINT:=0;
	RSP_SNODE: UINT:=0;
	RSP_TYPE: BYTE:=0;
	RSP_FREE: BYTE:=0;
	RSP_CONF: ULINT:=0; // variabile temporanea per la compressione 	
END_VAR

VAR
	iTemp1: INT;
	iTemp2: INT;
END_VAR


IF (init = FALSE) THEN	
	mngInit();
ELSE
	LOOP_COUNTER:= MAX_LOOP;
	//VERIFICA STATO BUS
	BUSSTATE:=CL2.GetBusState(stCanbus.stChannel.driver,ADR(eError));
	IF (BUSSTATE = CL2.BUSSTATE.BUSOFF) THEN
		CL2.ResetBusAlarm(stCanbus.stChannel.driver);
	END_IF
	
	// RICEZIONE DEL MESSAGGIO
	catchMessages();
	mngMessage();
	mngResponse();	
	
	//CICLO PER SVUOTARE IL BUFFER DI RICEZIONE
	WHILE ((LOOP_COUNTER > 0) AND (ctMsgLeft > 0)) DO 
		catchMessages();
		mngMessage();
		mngResponse();	
		LOOP_COUNTER:= LOOP_COUNTER-1;
	END_WHILE 

	// ***************** Gestione timer online ***************** //
	
	IF COMM_TIMER>0 THEN
		COMM_TIMER:=COMM_TIMER-1;
		grComm.bCommunicationActive:=TRUE;
	ELSE
		grComm.bCommunicationActive:=FALSE;
	END_IF
END_IF

METHOD PRIVATE mngInit
VAR_INPUT
END_VAR
IF stCanbus.bActive AND stCanbus.stChannel.bInitialized THEN
	registerReceiveMask(udiId:= grComm.uiProtocolMessageID, stCanBus:=stCanbus, receiveMask:= stReceiveMaks);
	init:= stReceiveMaks.bInitialized;
END_IF
END_METHOD

METHOD PRIVATE catchMessages
VAR_INPUT
END_VAR
// ***************** Cattura messaggi ***************** //

IF readMessage(stReceiveMask:=stReceiveMaks, byaReceivedData=> CAN_RX_BUFFER) > 0 THEN
	CAN_RX_COUNT:=CAN_RX_COUNT+1;
END_IF
END_METHOD

METHOD PRIVATE mngMessage
VAR_INPUT
END_VAR

VAR
	CMD_CONF: ULINT:=0; // variabile temporanea per l'estrazione 
	EEPROM_OP_RESULT: BOOL:= FALSE;
	GETSETVAR_OP_RESULT: BOOL:= FALSE;
END_VAR
// ***************** Elaborazione comando ***************** //

IF CAN_RX_COUNT > 0 THEN
	
	CAN_RX_COUNT:= CAN_RX_COUNT-1; 
	
	CMD_ADDR:= CAN_RX_BUFFER[1];
	CMD_ADDR:= SHL(CMD_ADDR, 8) OR CAN_RX_BUFFER[0];
	CMD_DATA:= CAN_RX_BUFFER[3];
	CMD_DATA:= SHL(CMD_DATA,8) OR CAN_RX_BUFFER[2];
		
	CMD_CONF:= CAN_RX_BUFFER[7];
	CMD_CONF:= SHL(CMD_CONF, 8) OR CAN_RX_BUFFER[6];
	CMD_CONF:= SHL(CMD_CONF, 8) OR CAN_RX_BUFFER[5];
	CMD_CONF:= SHL(CMD_CONF, 8) OR CAN_RX_BUFFER[4];
	
	CMD_SNODE:= ULINT_TO_UINT( SHR(CMD_CONF, 0) AND 16#003F );
	CMD_DNODE:= ULINT_TO_UINT( SHR(CMD_CONF, 6) AND 16#003F );
	CMD_PROG:= ULINT_TO_UINT( SHR(CMD_CONF, 12) AND 16#0FFF );
	CMD_FREE:= ULINT_TO_BYTE( SHR(CMD_CONF, 24) AND 16#000F );
	CMD_TYPE:= ULINT_TO_BYTE( SHR(CMD_CONF, 28) AND 16#000F );
	
	//CMD_DATA:= CMD_DATA AND LREAL_TO_UINT(EXPT(2, (CMD_DLEN+1)-1));	// Maschera del campo DATA in base alla lunghezza
		
	

	// Se il messaggio non è per me o non è valido exit
	IF ( (NOT(CMD_SNODE = CMD_DNODE) AND (CMD_DNODE = grComm.uiProtocolVirtualNode)) OR CMD_TYPE = grCommMessageType.HeartRateRequest ) THEN

		COMM_TIMER:= grComm.COMM_TIMER_RLD;
			
		// ____ Preimpostazione della risposta ____ //
		RSP_ADDR:= CMD_ADDR; 
		RSP_DATA:= 0;
		RSP_CONF:= 0;
		RSP_SNODE:= grComm.uiProtocolVirtualNode;
		RSP_DNODE:= CMD_SNODE;
		RSP_PROG:= CMD_PROG;
		RSP_FREE:= 0;
		RSP_TYPE:= INT_TO_BYTE(grCommMessageType.ErrorCode);  // fino a prova contraria
		
	
		// ____ Elaborazione comando ____ //
		CASE BYTE_TO_INT(CMD_TYPE) OF
			
			grCommMessageType.GetVariable:
				getsetVarCallback(VAR_ID:=CMD_ADDR, INPUT_VAL:=0, READ:=FALSE, VAR_RET => RSP_DATA, ESITO_OPERAZIONE=>GETSETVAR_OP_RESULT);
				IF GETSETVAR_OP_RESULT = TRUE THEN
					RSP_TYPE:= INT_TO_BYTE(grCommMessageType.ExitCode);
				END_IF
			
			grCommMessageType.SetVariable:
				getsetVarCallback(VAR_ID:=CMD_ADDR, INPUT_VAL:=CMD_DATA, READ:=TRUE, VAR_RET => RSP_DATA, ESITO_OPERAZIONE=>GETSETVAR_OP_RESULT);
				IF GETSETVAR_OP_RESULT = TRUE THEN
					RSP_TYPE:= INT_TO_BYTE(grCommMessageType.ExitCode);
				END_IF
			
			grCommMessageType.HeartRateRequest:
				RSP_TYPE:= INT_TO_BYTE(grCommMessageType.ExitCode);
			
			grCommMessageType.LoadFromEEPROM:
				readAllFromEEPROMCallback(ESITO_OPERAZIONE=>EEPROM_OP_RESULT);
				IF EEPROM_OP_RESULT = TRUE THEN
					RSP_TYPE:= INT_TO_BYTE(grCommMessageType.ExitCode);
				END_IF
			
			grCommMessageType.WriteToEEPROM:
				writeToEEPROMCallback(IGNORE_FLAG:=FALSE, ESITO_OPERAZIONE=>EEPROM_OP_RESULT);
				IF EEPROM_OP_RESULT = TRUE THEN
					RSP_TYPE:= INT_TO_BYTE(grCommMessageType.ExitCode);
				END_IF
					
			grCommMessageType.WriteAllToEEPROM:
				writeToEEPROMCallback(IGNORE_FLAG:=TRUE, ESITO_OPERAZIONE=>EEPROM_OP_RESULT);
				IF EEPROM_OP_RESULT = TRUE THEN
					RSP_TYPE:= INT_TO_BYTE(grCommMessageType.ExitCode);
				END_IF
					
			grCommMessageType.ApplyVariables:
				applyToRamCallback(ESITO_OPERAZIONE=>EEPROM_OP_RESULT);
				IF EEPROM_OP_RESULT = TRUE THEN
					RSP_TYPE:= INT_TO_BYTE(grCommMessageType.ExitCode);
				END_IF
			
			
			ELSE
				;// PASS
						
		END_CASE
		
		TX_COMM:= TRUE;
		
	ELSE	
		MISSED_COUNTER:=MISSED_COUNTER+1;
	END_IF	
	
	CMD_ADDR:= 0;
	CMD_DATA:= 0;
	CMD_CONF:= 0;
	CMD_SNODE:= 0;
	CMD_DNODE:= 0;
	CMD_PROG:= 0;
	CMD_FREE:= 0;
	CMD_TYPE:= 0;
	
	
END_IF
END_METHOD

METHOD PRIVATE mngResponse
VAR_INPUT
END_VAR

VAR
	TMP_NODE: UINT:= 0;
	stMessage: canMessage;
END_VAR
// ***************** Invio messaggio di risposta ***************** //

IF TX_COMM THEN
	
	// ____ Compressione data ____ //		
	TMP_NODE:= RSP_DNODE;
	TMP_NODE:= SHL(TMP_NODE, 6) OR RSP_SNODE;
	
	RSP_CONF:= (RSP_TYPE AND 16#0F);
	RSP_CONF:= SHL(RSP_CONF, 4) OR (RSP_FREE AND 16#0F);
	RSP_CONF:= SHL(RSP_CONF, 12) OR (RSP_PROG AND 16#0FFF);
	RSP_CONF:= SHL(RSP_CONF, 12) OR (TMP_NODE AND 16#0FFF);
	
	
	
	// ____ Invio messaggio ____ //
	
	CAN_TX_BUFFER[0] := UINT_TO_BYTE(SHR(RSP_ADDR, 0) AND 16#FF);	
	CAN_TX_BUFFER[1] := UINT_TO_BYTE(SHR(RSP_ADDR, 8) AND 16#FF);						
	CAN_TX_BUFFER[2] := UINT_TO_BYTE(SHR(RSP_DATA, 0) AND 16#FF);
	CAN_TX_BUFFER[3] := UINT_TO_BYTE(SHR(RSP_DATA, 8) AND 16#FF);
	CAN_TX_BUFFER[4] := ULINT_TO_BYTE(SHR(RSP_CONF, 0) AND 16#FF);	
	CAN_TX_BUFFER[5] := ULINT_TO_BYTE(SHR(RSP_CONF, 8) AND 16#FF);							
	CAN_TX_BUFFER[6] := ULINT_TO_BYTE(SHR(RSP_CONF, 16) AND 16#FF);	
	CAN_TX_BUFFER[7] := ULINT_TO_BYTE(SHR(RSP_CONF, 24) AND 16#FF);	
	
	stMessage.udiId:= grComm.uiProtocolMessageID;
	stMessage.byLength:= 8;
	stMessage.bExtended:= FALSE;
	stMessage.byaData:= CAN_TX_BUFFER;
	sendMessage(stCanBus:=stCanbus, stMessageToSend:= stMessage, Fault=> );
	
	CAN_TX_BUFFER[0]:= 0;
	CAN_TX_BUFFER[1]:= 0;
	CAN_TX_BUFFER[2]:= 0;
	CAN_TX_BUFFER[3]:= 0;
	CAN_TX_BUFFER[4]:= 0;
	CAN_TX_BUFFER[5]:= 0;
	CAN_TX_BUFFER[6]:= 0;
	CAN_TX_BUFFER[7]:= 0;
	TMP_NODE:= 0;
	RSP_CONF:= 0;	
	TX_COMM:= FALSE;
	
END_IF
END_METHOD

METHOD PRIVATE getsetVarCallback: UINT

VAR_INPUT
	VAR_ID: UINT:= 0;
	INPUT_VAL: UINT:= 0; 
	READ: BOOL; // se == 0 significa GET_VAR, altrimenti SET_VAR
END_VAR


VAR_OUTPUT	
	VAR_RET: UINT:= 0;
	ESITO_OPERAZIONE: BOOL:= FALSE;
END_VAR
ESITO_OPERAZIONE:= TRUE;

IF VAR_ID > 0 AND VAR_ID <= grComm.uiVariablesMaxIndex THEN
	
	IF READ = FALSE AND grComm.staVariables[VAR_ID].accessRights <> grCommAccessRight.NoAccess THEN
		VAR_RET:= grComm.staVariables[VAR_ID].uiValue;
	ELSIF grComm.staVariables[VAR_ID].accessRights = grCommAccessRight.ReadWrite THEN
		IF (INPUT_VAL < grComm.staVariables[VAR_ID].uiLowerValidValue OR INPUT_VAL > grComm.staVariables[VAR_ID].uiHigherValidValue) THEN
			INPUT_VAL:= grComm.staVariables[VAR_ID].uiDefaultValue;
		END_IF
		grComm.staVariables[VAR_ID].uiValue:= INPUT_VAL;
		grComm.staVariables[VAR_ID].status:= grCommVariableStatus.ModifiedByRemote;
	ELSE
		ESITO_OPERAZIONE:= FALSE;
		grComm.staVariables[VAR_ID].status:= grCommVariableStatus.Error;
	END_IF
	
ELSE
	(* Requested ID is invalid *)
	ESITO_OPERAZIONE:= FALSE;
END_IF
END_METHOD

METHOD PRIVATE applyToRamCallback: BOOL;
VAR_INPUT
END_VAR

VAR_OUTPUT
	ESITO_OPERAZIONE: BOOL:= FALSE;
END_VAR
grComm.bTriggerApplyToRAM:= TRUE;
ESITO_OPERAZIONE:= TRUE;
END_METHOD

METHOD PRIVATE readAllFromEEPROMCallback: BOOL;
VAR_INPUT
END_VAR


VAR_OUTPUT
	ESITO_OPERAZIONE: BOOL:= FALSE;
END_VAR

VAR
	uiVarIterator: UINT;
END_VAR
grComm.bTriggerReadFromEEPROM:= TRUE;

ESITO_OPERAZIONE:= TRUE;
END_METHOD

METHOD PRIVATE writeToEEPROMCallback: BOOL;
VAR_INPUT
	IGNORE_FLAG: BOOL:= FALSE;
END_VAR

VAR_OUTPUT
	ESITO_OPERAZIONE: BOOL:= FALSE;
END_VAR
applyToRamCallback();
grComm.bTriggerWriteAllToEEPROM:= (IGNORE_FLAG);
grComm.bTriggerWriteToEEPROM:= (NOT IGNORE_FLAG);

ESITO_OPERAZIONE:= TRUE;
END_METHOD

METHOD PUBLIC applyToRAM
VAR
	uiVarIterator: UINT;
END_VAR
FOR uiVarIterator:= 1 TO grcomm.uiVariablesMaxIndex BY 1 DO
	IF mngCommCan.isVariableValid(grcomm.staVariables[uiVarIterator]) AND grcomm.staVariables[uiVarIterator].status = grCommVariableStatus.ModifiedByRemote THEN
		grcomm.staVariables[uiVarIterator].pointerToSystemVar^:= grcomm.staVariables[uiVarIterator].uiValue;
		grcomm.staVariables[uiVarIterator].status:= grCommVariableStatus.Pristine;
	END_IF
END_FOR
END_METHOD

METHOD PUBLIC isVariableValid : BOOL
VAR_INPUT
	variable: grCommVar;
END_VAR
isVariableValid:= (
	variable.pointerToSystemVar > 0
	);
END_METHOD

METHOD PUBLIC initializeVariable : grCommVar
VAR_INPUT
	pointerToSystemVar: POINTER TO UINT;
	accessRights: grCommAccessRight;
	uiDefaultValue: UINT;
	uiLowerValidValue: UINT;
	uiHigherValidValue: UINT;
END_VAR

VAR 
	newVar: grCommVar;
	tmpVal: UINT;
END_VAR
newVar.pointerToSystemVar:= pointerToSystemVar;
newVar.accessRights:= accessRights;
newVar.uiDefaultValue:= uiDefaultValue;
newVar.uiLowerValidValue:= uiLowerValidValue;
newVar.uiHigherValidValue:= uiHigherValidValue;

tmpVal:= pointerToSystemVar^;
IF(tmpVal < uiLowerValidValue OR tmpVal > uiHigherValidValue) THEN
	tmpVal:= uiDefaultValue;
	pointerToSystemVar^:= uiDefaultValue;
END_IF
newVar.uiValue:= tmpVal;

initializeVariable:= newVar;
END_METHOD

END_PROGRAM

// Device/Application/Modules/Canbus/Functions/registerReceiveMask
// This PRG contains non safety-related code.
// The following attribute is autogenerated. Do not remove.
{attribute 'location':='16#800'}
PROGRAM registerReceiveMask
VAR_INPUT
	stCanBus: canBus;
	udiId: UDINT:= 0;
	udiCobIdMask: UDINT:= 16#1FFFFFFF;
	xExtended: BOOL:= TRUE;
END_VAR
VAR_IN_OUT
	receiveMask: canReceiveMask;
END_VAR

IF (udiId > 0) THEN	
	receiveMask.udiId:= udiId;
	receiveMask.udiCobIdMask:= udiCobIdMask;
	checkReceiveMaskInitialization(stCan:= stCanBus.stChannel, stReceiveMask:= receiveMask);
	receiveMask.bActive:= TRUE;
END_IF

END_PROGRAM

// Device/Application/Modules/Canbus/Functions/checkReceiveMaskInitialization
// This PRG contains non safety-related code.
// The following attribute is autogenerated. Do not remove.
{attribute 'location':='16#800'}
PROGRAM checkReceiveMaskInitialization
VAR_INPUT
	stCan: can;
END_VAR
VAR_IN_OUT
	stReceiveMask: canReceiveMask;
END_VAR
VAR	
	cobIdMask: CL2.CL2I.COBID:= 16#1FFFFFFF; 
	xRTRValue: BOOL:= FALSE;
	xRTRMask: BOOL:= FALSE;
	x29BitIdValue: BOOL:= FALSE; 
	x29BitIdMask: BOOL:= FALSE;
	xTransmitValue: BOOL:= FALSE; 
	xTransmitMask: BOOL:= TRUE;
	xAlwaysNewest: BOOL:= FALSE; 
	eEvent: CL2.CB.EVENT:= 0;
	xEnableSyncWindow: BOOL:= FALSE; 
END_VAR

IF (stCan.bInitialized) AND (stReceiveMask.stCAAMask = CL2.CAA.gc_hINVALID) THEN	
	stReceiveMask.stCAAMask := CL2.CreateMaskReceiver(
		hDriver := stCan.driver, 
		cobIdValue := stReceiveMask.udiId, 
		cobIdMask := stReceiveMask.udiCobIdMask, 
		xRTRValue := xRTRValue, 
		xRTRMask := xRTRMask, 
		x29BitIdValue := x29BitIdValue, 
		x29BitIdMask := x29BitIdMask, 
		xTransmitValue := xTransmitValue, 
		xTransmitMask := xTransmitMask, 
		xAlwaysNewest := xAlwaysNewest, 
		eEvent := eEvent,
		xEnableSyncWindow := xEnableSyncWindow, 
		peError := 0
	);
	
	(*hReceiver := CL2.CreateMaskReceiver(hDriver := canbus.stChannel.driver,
					cobIdValue := 16#18FFFF00, 
					cobIdMask := 16#1F0000FF, 
					xRTRValue := FALSE, //no RTR messages
					xRTRMask := TRUE, //activate RTR filter ==> xRTRValue will be checked
					x29BitIdValue := TRUE, //no 29 bit CAN messages
					x29BitIdMask := TRUE, //activate 29 bit filter ==> x29BitIdValue will be checked
					xTransmitValue := FALSE, //only receive messages, no transmit message loopback
					xTransmitMask := TRUE, //activate transmit mask filter ==> xTransmitValue will be checked
					xAlwaysNewest := FALSE, //FALSE := receiver with queue; TRUE: only newest message
					eEvent := 0, //no receive event
					xEnableSyncWindow := FALSE, //not implemented
					peError := ADR(fault) //optional pointer to error
				);*)
END_IF

IF stReceiveMask.stCAAMask <> CL2.CAA.gc_hINVALID THEN
	stReceiveMask.bInitialized:= TRUE;
END_IF

END_PROGRAM

// Device/Application/Modules/Canbus/Functions/readMessage
// This PRG contains non safety-related code.
// The following attribute is autogenerated. Do not remove.
{attribute 'location':='16#800'}
FUNCTION readMessage: INT;
VAR_IN_OUT
	stReceiveMask: canReceiveMask;
END_VAR
VAR_OUTPUT
	readCount: INT;
	byaReceivedData: ARRAY [0..7] OF BYTE;
END_VAR
VAR	
	iCounter: INT:= 0;
	iReceivedCount: INT:= 0;
	stReceivedMessage: CL2.CAA.HANDLE := CL2.CAA.gc_hINVALID;
	stReceiveError: CL2.ERROR;
	usiTmpData: ARRAY [0..7] OF USINT;
END_VAR

iReceivedCount:= 0;
IF stReceiveMask.bActive THEN
	stReceivedMessage:= CL2.Read(hReceiverId:=stReceiveMask.stCAAMask, pctMsgLeft:=ADR(stReceiveMask.stMessagesLeft), peError:=ADR(stReceiveError));
		
	IF stReceivedMessage <> CL2.CAA.gc_hINVALID THEN
		usiTmpData:= CL2.GetMessageDataPointer(hMessage:=stReceivedMessage, peError:=ADR(stReceiveError))^;
		FOR iCounter:=0 TO 7 BY 1 DO
			byaReceivedData[iCounter]:= USINT_TO_BYTE(usiTmpData[iCounter]);
		END_FOR
		CL2.FreeMessage(hMessage:= stReceivedMessage);
		iReceivedCount:= 1;
	END_IF
END_IF
readCount:= iReceivedCount;

// Per l'uso come function
readMessage:= readCount;

END_FUNCTION

// Device/Application/Modules/Canbus/Functions/sendMessage
// This PRG contains non safety-related code.
// The following attribute is autogenerated. Do not remove.
{attribute 'location':='16#800'}
PROGRAM sendMessage

VAR_INPUT
	stCanBus: canBus;
	stMessageToSend: canMessage;
END_VAR

VAR_OUTPUT
	Fault : CL2.ERROR;
END_VAR

VAR
	stCan: can;
	EXT : BOOL;
	ID : CL2.CL2I.COBID;
	LEN : USINT;
	TX_pointer	: POINTER TO CL2.CL2I.DATA;
	DRIVER : CL2.CAA.HANDLE;
	
	
	hTxMsg : CL2.CAA.HANDLE := CL2.CAA.gc_hINVALID;
	x29Bit : BOOL;
	xRTR : BOOL;
	xTxFrame : BOOL;
	eError : CL2.ERROR;
	pTxData : POINTER TO CL2.CL2I.DATA;
	diMsgRecv: DINT;
	i : INT;
END_VAR

stCan:= stCanBus.stChannel;
EXT:=stMessageToSend.bExtended;
ID:= stMessageToSend.udiId;
LEN:= stMessageToSend.byLength; 
TX_pointer:= ADR(stMessageToSend.byaData); 
DRIVER:= stCan.driver;

checkBusState(stCan:= stCan);		
		
IF(TRUE (*ID > 0*)) THEN		
	IF(LEN > 8) THEN
		LEN:= 8;
	END_IF
	hTxMsg := CL2.CreateMessage(
		hDriver := DRIVER, 
		cobID := ID, 
		usiLength := LEN, 
		xRTR := xRTR, 
		x29BitID := EXT, 
		peError := ADR(eError));
		
	IF hTxMsg <> CL2.CAA.gc_hINVALID THEN
		pTxData := CL2.GetMessageDataPointer(hMessage := hTxMsg, peError := ADR(eError));
		IF pTxData <> CL2.CAA.gc_pNULL AND LEN <> 0 THEN
			FOR i := 0 TO LEN - 1 DO
				pTxData^[i] := TX_pointer^[i];
			END_FOR
		END_IF
		eError := CL2.Write(hDriver := DRIVER, hMessage := hTxMsg, usiPriority := 1, xEnableSyncWindow := FALSE);
		IF eError <> CL2.ERROR.NO_ERROR THEN
			CL2.FreeMessage(hMessage := hTxMsg);
		END_IF
		hTxMsg := CL2.CAA.gc_hINVALID;
		pTxData := CL2.CAA.gc_pNULL;
		Fault:= stCan.transmitError;
	END_IF
END_IF

END_PROGRAM

// Device/Application/Modules/Canbus/Functions/checkBusState
// This PRG contains non safety-related code.
// The following attribute is autogenerated. Do not remove.
{attribute 'location':='16#800'}
PROGRAM checkBusState
VAR_INPUT
	stCan: can;
END_VAR
VAR
	stResetResult: CL2.ERROR:= CL2.ERROR.INVALID_HANDLE;
END_VAR

IF (stCan.bInitialized) AND	(stCan.busStatus <> CL2.BUSSTATE.ERR_FREE) AND (stCan.busStatus <> CL2.BUSSTATE.ACTIVE) THEN
	stResetResult:= CL2.ResetBusAlarm(hDriver:= stCan.driver);
END_IF

END_PROGRAM

// Device/Application/Program logic/Tasks/CanComunication
PROGRAM CanComunication
VAR CONSTANT
	uiNode: UINT:= 16#10;
	displayNode: BYTE:= 16#DD;
END_VAR
VAR
	xInitialized: BOOL:= FALSE;
	stCanbusPC: canBus;	
	stCanbusETSDN: canBus;	
	
	uiSendVariablesTimerMs: UINT;
	uiStartupTimerMs: UINT:= 60000;
	
	FlasherMsgConf: canReceiveMask;
	FlasherMsgComEtsdn: canReceiveMask;
	FlasherMsgComEtsOne: canReceiveMask;	
	
	displayMsgIO: canReceiveMask;
	
	etsdnIOMsg1Mask: canReceiveMask;
	etsdnIOMsg2Mask: canReceiveMask;
	etsdnAccMsgMask: canReceiveMask;
	
	
	uiAntiBumpTimer: UINT:= 0;
	uiAntiBumpIntervalMs: UINT:= 100;
	uiDisplayMsgIOTimerMs: UINT;
	
	byMsgSendStep: BYTE:= 0;
	
	

END_VAR

IF NOT xInitialized THEN
	stCanbusPC:= fieldbus.can[4];
	stCanbusETSDN := fieldbus.can[4];
	xInitialized:= initialize();
	
ELSE
	IF uiSendVariablesTimerMs = 0 THEN
		uiSendVariablesTimerMs:= 100;
		sendVariablesDisplay();
		SendVariablesFromEtsdn(RxFlasher.systemUnderTest);
	ELSE
		Utils.decrementUINT(uiSendVariablesTimerMs, 10);
	END_IF
	receiveVariables();
	Utils.decrementUINT(uiStartupTimerMs, 10);
END_IF

METHOD PRIVATE sendVariablesDisplay
VAR
	msg: canMessage;
	rTmpAirPressure: REAL;
	uiTmpSpeed: UINT;
	

END_VAR
msg.bExtended:= FALSE;

msg.udiId:= 16#280;
msg.byLength:= 8;

msg.byaData[0].0:= system.xTestRunning;
msg.byaData[0].1:= system.xTestResultValid;
msg.byaData[0].2:= system.xTestResult;
msg.byaData[0].3:= system.xCanTestResult;
msg.byaData[0].4:= system.xDigitalInTestResult;
msg.byaData[0].5:= system.xAnalogInTestResult;
msg.byaData[0].6:= system.xPowerTestResult;
msg.byaData[0].7:= system.x5VOutTestResult;
msg.byaData[1].0:= system.xAccelerometerTestResult;

msg.byaData[1].1:= (system.iAccTestStep = 0);
msg.byaData[1].2:= (system.iAccTestStep = 1);
msg.byaData[1].3:= (system.iAccTestStep = 2);

msg.byaData[1].4:= system.xReleTestResult;

msg.byaData[1].5:= EtsdnVar.xOnline OR ETSDN_Test_PRG.iTestStep = 13;

msg.byaData[2]:= system.byTestPercentage;
msg.byaData[3]:= INT_TO_BYTE(ETSDN_Test_PRG.iTestStep+1);
		
sendMessage(stCanBus:= stCanbusPC, stMessageToSend:= msg);
END_METHOD

METHOD PRIVATE receiveVariables
VAR
	byaData: ARRAY[0..7] OF BYTE;
	
	byaDataEtsdn: ARRAY[0..7] OF BYTE;
	wTmp: WORD;
	dwTmp:DWORD;
	pTmp: POINTER TO DWORD;
	
END_VAR

VAR_STAT
	uiFlasherMsgConfTimerMs: UINT;
	uiFlasherMsgComEtsdnTimerMs: UINT;
	uiFlasherMsgComEtsOneTimerMs: UINT;
	uiETSDNOnlineTimerMs: UINT;
END_VAR
(* Ricezione da Flasher il selettore della centralina da collaudare *)
WHILE readMessage(stReceiveMask:= FlasherMsgConf, byaReceivedData=> byaData) > 0 DO
	RxFlasher.systemUnderTest:= byaData[0];
 
	uiFlasherMsgConfTimerMs:= 1000;
END_WHILE	
Utils.decrementUINT(uiFlasherMsgConfTimerMs, 10);

(* Ricezione da Flasher il test da effettuare all'ETSDN *)
WHILE readMessage(stReceiveMask:= FlasherMsgComEtsdn, byaReceivedData=> byaData) > 0 DO
	EtsdnVar.cmdTest:= byaData[0];
    EtsdnVar.xRL1 := byaData[1].0;
	EtsdnVar.xRL2 := byaData[1].1;
	EtsdnVar.xRL3 := byaData[1].2;
	EtsdnVar.xPwrSupplyRL1 := byaData[1].3;
	EtsdnVar.xPwrSupplyRL2 := byaData[1].4; 
	EtsdnVar.xPwrSupplyRL3 := byaData[1].5;					(*Ricevo i messaggi da Flash per decidere che test effetturare ETSDN*)
	
	EtsdnVar.xCycle10V := byaData[1].6;
	
	EtsdnVar.xPwrSupplyIP1 := byaData[2].0; 
	EtsdnVar.xPwrSupplyIP2 := byaData[2].1;
	EtsdnVar.xPwrSupplyIN1 := byaData[2].2;
	EtsdnVar.xPwrSupplyIN2 := byaData[2].3;
	
	uiFlasherMsgComEtsdnTimerMs:= 1000;
END_WHILE	
Utils.decrementUINT(uiFlasherMsgComEtsdnTimerMs, 10);

(* Ricezione da Flasher il test da effettuare all'Etsone *)
WHILE readMessage(stReceiveMask:= FlasherMsgComEtsOne, byaReceivedData=> byaData) > 0 DO
	EtsOneVar.cmdTest:= byaData[0];
	EtsOneVar.xOneRL1 := byaData[1].0;
    EtsOneVar.xOneRL2:= byaData[1].1;						
	EtsOneVar.xOneIP1 := byaData[1].2;								(*Ricevo i messaggi da Flash per decidere che test effetturare *)
	EtsOneVar.xOneIP2 := byaData[1].3;
	EtsOneVar.xOneIP3 := byaData[1].4;
	EtsOneVar.xCycleOneIP4 := byaData[1].5;
	EtsOneVar.dwOne5V := byaData[4];
	
	uiFlasherMsgComEtsOneTimerMs:= 1000;
END_WHILE	
Utils.decrementUINT(uiFlasherMsgComEtsOneTimerMs, 10);

CASE RxFlasher.systemUnderTest OF 
	
    1:  // etsdn
		WHILE readMessage(stReceiveMask:= etsdnIOMsg1Mask, byaReceivedData=> byaDataEtsdn) > 0 DO
		
			EtsdnVar.xIP1:= byaDataEtsdn[0].0;
			EtsdnVar.xIP2:= byaDataEtsdn[0].1;
			EtsdnVar.xIN1:= byaDataEtsdn[0].2;
			EtsdnVar.xIN2:= byaDataEtsdn[0].3;
			
			pTmp:= ADR(EtsdnVar.rSupplyVoltage);
			pTmp^:= (byaDataEtsdn[4] OR SHL(BYTE_TO_DWORD(byaDataEtsdn[5]), 8) OR SHL(BYTE_TO_DWORD(byaDataEtsdn[6]), 16) OR SHL(BYTE_TO_DWORD(byaDataEtsdn[7]), 24));
			
		 	EtsdnVar.msgRx_01 := byaDataEtsdn;
			
			uiETSDNOnlineTimerMs:= 1000;
		END_WHILE	
		
		
		WHILE readMessage(stReceiveMask:= etsdnIOMsg2Mask, byaReceivedData=> byaDataEtsdn) > 0 DO
			pTmp:= ADR(EtsdnVar.rIP3);
			pTmp^:= (byaDataEtsdn[0] OR SHL(BYTE_TO_DWORD(byaDataEtsdn[1]), 8) OR SHL(BYTE_TO_DWORD(byaDataEtsdn[2]), 16) OR SHL(BYTE_TO_DWORD(byaDataEtsdn[3]), 24));
		
			pTmp:= ADR(EtsdnVar.rAI);
			pTmp^:= (byaDataEtsdn[4] OR SHL(BYTE_TO_DWORD(byaDataEtsdn[5]), 8) OR SHL(BYTE_TO_DWORD(byaDataEtsdn[6]), 16) OR SHL(BYTE_TO_DWORD(byaDataEtsdn[7]), 24));
		 
			EtsdnVar.msgRx_02 := byaDataEtsdn;
			uiETSDNOnlineTimerMs:= 1000;
		END_WHILE	
		
		
		WHILE readMessage(stReceiveMask:= etsdnAccMsgMask, byaReceivedData=> byaDataEtsdn) > 0 DO
			wTmp:= byaDataEtsdn[0] OR SHL(BYTE_TO_WORD(byaDataEtsdn[1]), 8);
			EtsdnVar.rY:= INT_TO_REAL(WORD_TO_INT(wTmp)) * 0.000244140625;
			wTmp:= byaDataEtsdn[2] OR SHL(BYTE_TO_WORD(byaDataEtsdn[3]), 8);
			EtsdnVar.rX:= INT_TO_REAL(WORD_TO_INT(wTmp)) * 0.000244140625;
			wTmp:= byaDataEtsdn[6] OR SHL(BYTE_TO_WORD(byaDataEtsdn[7]), 8);
			EtsdnVar.rZ:= INT_TO_REAL(WORD_TO_INT(wTmp)) * 0.000244140625;
		 
			EtsdnVar.msgRx_03 := byaDataEtsdn;
			uiETSDNOnlineTimerMs:= 1000;
		END_WHILE
		
		Utils.decrementUINTTimer(uiETSDNOnlineTimerMs);
		
		EtsdnVar.xOnline:= (uiETSDNOnlineTimerMs > 0);
		
		IF NOT EtsdnVar.xOnline THEN
			EtsdnVar.rY:= 0;
			EtsdnVar.rX:= 0;
			EtsdnVar.rZ:= 0;
			EtsdnVar.rIP3:= 0;
			EtsdnVar.rAI:= 0;
			EtsdnVar.xIP1:= 0;
			EtsdnVar.xIP2:= 0;
			EtsdnVar.xIN1:= 0;
			EtsdnVar.xIN2:= 0;
		END_IF
		
	2: 

			
END_CASE
Utils.decrementUINT(uiAntiBumpTimer, 10);
Utils.decrementUINT(uiDisplayMsgIOTimerMs, 10);


IF uiFlasherMsgConfTimerMs = 0 THEN
	RxFlasher.systemUnderTest := 0;
END_IF

IF uiFlasherMsgConfTimerMs = 0 THEN
	EtsdnVar.cmdTest := 0;
END_IF
END_METHOD

METHOD PRIVATE initialize: BOOL;
VAR
	xRet: BOOL;
END_VAR
initialize:= FALSE;
IF stCanbusPC.bActive AND stCanbusPC.stChannel.bInitialized THEN
	registerReceiveMask(udiId:= 16#180, stCanBus:=stCanbusPC, receiveMask:= FlasherMsgConf); // ricevuto da PC
	
	registerReceiveMask(udiId:= 16#280, stCanBus:=stCanbusPC, receiveMask:= FlasherMsgComEtsOne);  // ricevuto da PC  
	
	registerReceiveMask(udiId:= 16#380, stCanBus:=stCanbusPC, receiveMask:= FlasherMsgComEtsdn);    // ricevuto da PC

	

END_IF


IF stCanbusETSDN.bActive AND stCanbusETSDN.stChannel.bInitialized THEN

	registerReceiveMask(udiId:= 16#20001, stCanBus:=stCanbusETSDN, receiveMask:= etsdnIOMsg1Mask);  // ricevuto da etsdn
	registerReceiveMask(udiId:= 16#20002, stCanBus:=stCanbusETSDN, receiveMask:= etsdnIOMsg2Mask);  // ricevuto da etsdn
	registerReceiveMask(udiId:= 16#20003, stCanBus:=stCanbusETSDN, receiveMask:= etsdnAccMsgMask);  // ricevuto da etsdn
	

END_IF

initialize:= FlasherMsgConf.bInitialized AND FlasherMsgComEtsOne.bInitialized AND FlasherMsgComEtsdn.bInitialized AND etsdnIOMsg1Mask.bInitialized AND etsdnIOMsg2Mask.bInitialized AND etsdnAccMsgMask.bInitialized;
END_METHOD

METHOD PRIVATE SendVariablesFromEtsdn
VAR
	msg: canMessage;
	arrayNullo : ARRAY[0..7] OF BYTE := [0, 0, 0, 0, 0, 0,  0, 0];
	uVarTemp1 : UINT := 0;
	uVarTemp2 : UINT := 0;
	uVarTemp3 : UINT := 0;
	uVarTemp4 : UINT := 0;
END_VAR

VAR_INPUT
	typeOfTest : byte;
END_VAR
CASE typeOfTest OF
	1:	//ETSDN
	    (* Messaggio di *)
		msg.bExtended:= FALSE;
		
		msg.bExtended:= TRUE;
		msg.udiId:= 16#10000;
		msg.byLength:= 8;
		
		msg.byaData[0].0:= EtsdnVar.xRL1;
		msg.byaData[0].1:= EtsdnVar.xRL2;
		msg.byaData[0].2:= EtsdnVar.xRL3;
		sendMessage(stCanBus:= stCanbusPC, stMessageToSend:= msg);
		sendMessage(stCanBus:= stCanbusETSDN, stMessageToSend:= msg);
		
		
		msg.udiId:= 16#10001;
		uVarTemp1 := DWORD_TO_UINT(sysIO.analogInput.ecuK15_p207.dwValue/100);
		msg.byaData[1] := UINT_TO_BYTE(SHL(uVarTemp1,0));
		msg.byaData[0] := UINT_TO_BYTE(SHL(uVarTemp1,8));
		
		uVarTemp2 := DWORD_TO_UINT(sysIO.digitalOutput.etsPower_p177.wCurrent/100);
		msg.byaData[3] := UINT_TO_BYTE(SHL(uVarTemp2,0));
		msg.byaData[2] := UINT_TO_BYTE(SHL(uVarTemp2,8));
		
		uVarTemp3 := DWORD_TO_UINT(sysIO.analogInput.ets5V_p131.dwValue /100);
		msg.byaData[5] := UINT_TO_BYTE(SHL(uVarTemp3,0));
		msg.byaData[4] := UINT_TO_BYTE(SHL(uVarTemp3,8));
		
		msg.byaData[6] := 0;
		msg.byaData[7] := 0;
		
	
		sendMessage(stCanBus:= stCanbusPC, stMessageToSend:= msg);
		
		msg.udiId:= 16#10002;
		uVarTemp1 := DWORD_TO_UINT(sysIO.digitalOutput.etsRele_p183.wCurrent);
		msg.byaData[0] := UINT_TO_BYTE(SHL(uVarTemp1,0));
		msg.byaData[1] := UINT_TO_BYTE(SHL(uVarTemp1,8));
		
		uVarTemp2 := DWORD_TO_UINT(sysIO.digitalOutput.etsRele_p186.wCurrent);
		msg.byaData[2] := UINT_TO_BYTE(SHL(uVarTemp2,0));
		msg.byaData[3] := UINT_TO_BYTE(SHL(uVarTemp2,8));
		
		uVarTemp3 := DWORD_TO_UINT(sysIO.digitalOutput.etsRele_p180.wCurrent);
		msg.byaData[4] := UINT_TO_BYTE(SHL(uVarTemp3,0));
		msg.byaData[5] := UINT_TO_BYTE(SHL(uVarTemp3,8));
		
		msg.byaData[6] := 0;
		msg.byaData[7] := 0;
		
		sendMessage(stCanBus:= stCanbusPC, stMessageToSend:= msg);
		
		msg.udiId:= 16#20001;
		msg.byaData := EtsdnVar.msgRx_01;
		sendMessage(stCanBus:= stCanbusPC, stMessageToSend:= msg);
		
		
		
		msg.udiId:= 16#20002;
		msg.byaData := EtsdnVar.msgRx_02;
		sendMessage(stCanBus:= stCanbusPC, stMessageToSend:= msg);

		
		
		msg.udiId:= 16#20003;
		msg.byaData := EtsdnVar.msgRx_03;
		sendMessage(stCanBus:= stCanbusPC, stMessageToSend:= msg);
		
	2: //ETSONE
		

		msg.bExtended:= FALSE;
		
		msg.bExtended:= TRUE;
		msg.udiId:= 16#3001;
		msg.byLength:= 8;
		
		msg.byaData[0].1 := EtsOneVar.xOneRL1;
		msg.byaData[0].2 := EtsOneVar.xOneRL2;
		msg.byaData[0].3 := EtsOneVar.xOneIP1;
		msg.byaData[0].4 := EtsOneVar.xOneIP2;
		msg.byaData[0].5 := EtsOneVar.xOneIP3;
		msg.byaData[0].6 := EtsOneVar.xCycleOneIP4;
		
		msg.byaData[1]:= DWORD_TO_BYTE(sysIO.analogInput.ecuK15_p207.dwValue/100);
		msg.byaData[2]:= WORD_TO_BYTE(sysIO.digitalOutput.etsonePower_p153.wCurrent);
		msg.byaData[3]:= DWORD_TO_BYTE(sysIO.analogInput.etsone5V_107.dwValue /1000);
		
		msg.byaData[4] := WORD_TO_BYTE(EtsOneVar.rPwrSupplyOneRL1);
		msg.byaData[5]:= WORD_TO_BYTE(EtsOneVar.rPwrSupplyOneRL2);
		
		sendMessage(stCanBus:= stCanbusPC, stMessageToSend:= msg);
		
		
		
		

END_CASE
END_METHOD

METHOD PRIVATE SendVariablesFromEtsOne
VAR
	msg: canMessage;
	arrayNullo : ARRAY[0..7] OF BYTE := [0, 0, 0, 0, 0, 0,  0, 0];
END_VAR

VAR_INPUT
	typeOfTest : byte;
END_VAR
CASE typeOfTest OF
	1:
	    (* Messaggio da Plc a ETSDN *)
		msg.bExtended:= FALSE;
		
		msg.bExtended:= TRUE;
		msg.udiId:= 16#10000;
		msg.byLength:= 8;
		
		msg.byaData[0].0:= EtsdnVar.xRL1;
		msg.byaData[0].1:= EtsdnVar.xRL2;
		msg.byaData[0].2:= EtsdnVar.xRL3;
		sendMessage(stCanBus:= stCanbusPC, stMessageToSend:= msg);

		
		
	    (* Messaggio da Plc a ETSDN *)
		msg.bExtended:= FALSE;
		
		msg.bExtended:= TRUE;
		msg.udiId:= 16#10000;
		msg.byLength:= 8;
		
		msg.byaData[0].0:= EtsdnVar.xRL1;
		msg.byaData[0].1:= EtsdnVar.xRL2;
		msg.byaData[0].2:= EtsdnVar.xRL3;
		sendMessage(stCanBus:= stCanbusPC, stMessageToSend:= msg);
	
	// 2:
	
END_CASE
END_METHOD

END_PROGRAM

// Device/Application/Modules/Utils/Utils
PROGRAM Utils

VAR CONSTANT
	PWM_ON : WORD :=65000;
	PWM_OFF : WORD :=0;
END_VAR

VAR
	linTrafo: LIN_TRAFO;
END_VAR

METHOD decrementUINT
VAR_IN_OUT
	input: UINT;
END_VAR
VAR_INPUT
	step: UINT;
END_VAR
IF(step > input) THEN 
	input:= 0;
ELSE
	input:= input - step;
END_IF
END_METHOD

METHOD PUBLIC bytesToUInt16 : UINT
VAR_INPUT
	mostSignificantByte: BYTE;
	leastSignificantByte: BYTE;
END_VAR
bytesToUInt16:= SHL(BYTE_TO_UINT(mostSignificantByte), 8) OR leastSignificantByte;
END_METHOD

METHOD PUBLIC toggle
VAR_IN_OUT
	bValue: BOOL;
END_VAR
bValue:= NOT bValue;
END_METHOD

METHOD PUBLIC isNaN: BOOL
VAR_INPUT
	rTest: REAL;
END_VAR
isNaN:= NOT(rTest = rTest);
END_METHOD

METHOD PUBLIC updateValueFiltered : REAL
VAR_INPUT
	rCurrentValue: REAL;
	rNewValue: REAL;
	rFilterConstant: REAL;
END_VAR

VAR
	rFilteredValue: REAL;
END_VAR
rFilteredValue:= (rCurrentValue * rFilterConstant) + (rNewValue * (1 - rFilterConstant));
updateValueFiltered:= rFilteredValue;
END_METHOD

METHOD PUBLIC bytesToInt16 : INT
VAR_INPUT
	mostSignificantByte: BYTE;
	leastSignificantByte: BYTE;
END_VAR
bytesToInt16:= WORD_TO_INT(SHL(BYTE_TO_WORD(mostSignificantByte), 8) OR leastSignificantByte);
END_METHOD

METHOD decrementUDINT
VAR_IN_OUT
	input: UDINT;
END_VAR
VAR_INPUT
	step: UDINT;
END_VAR
IF(step > input) THEN 
	input:= 0;
ELSE
	input:= input - step;
END_IF
END_METHOD

METHOD PUBLIC boolToPWMDutyCycle : WORD
VAR_INPUT
	bEnable: BOOL;
END_VAR
IF bEnable THEN
	boolToPWMDutyCycle:= PWM_ON;
ELSE
	boolToPWMDutyCycle:= PWM_OFF;	
END_IF
END_METHOD

METHOD PUBLIC linearize: REAL
VAR_INPUT
	rIn: REAL;
	rInMin: REAL;
	rInMax: REAL;
	rOutMin: REAL;
	rOutMax: REAL;
END_VAR

VAR_OUTPUT
	xError: BOOL;
END_VAR

VAR
	rOut: REAL;
END_VAR
IF rIn < rInMin THEN rIn:= rInMin; END_IF
IF rIn > rInMax THEN rIn:= rInMax; END_IF

linTrafo(
	IN:= rIn,
	IN_MIN:= rInMin,
	IN_MAX:= rInMax,
	OUT_MIN:= rOutMin,
	OUT_MAX:= rOutMax,
	OUT=> rOut,
	ERROR=> xError
);

linearize:= rOut;
END_METHOD

METHOD PUBLIC bytesToUReal16 : REAL
VAR_INPUT
	mostSignificantByte: BYTE;
	leastSignificantByte: BYTE;
END_VAR
bytesToUReal16:= bytesToUInt16(mostSignificantByte, leastSignificantByte);
END_METHOD

METHOD PUBLIC bytesToUDInt32 : UDINT
VAR_INPUT
	byte0: BYTE;
	byte1: BYTE;
	byte2: BYTE;
	byte3: BYTE;
END_VAR
bytesToUDInt32:= SHL(BYTE_TO_UDINT(byte3), 24) OR SHL(BYTE_TO_UDINT(byte2), 16) OR SHL(BYTE_TO_UDINT(byte1), 8) OR byte0;
END_METHOD

METHOD incrementUINT
VAR_IN_OUT
	input: UINT;
END_VAR
VAR_INPUT
	step: UINT;
END_VAR
IF(step >= (16#FFFF - step)) THEN 
	input:= 16#FFFF;
ELSE
	input:= input + step;
END_IF
END_METHOD

METHOD PUBLIC getCurrentTaskCycleTime : DWORD // returns caller task interval in microseconds
VAR
    dwCycleTimeMainTask, dwCycleTimeSecTask    :    DWORD;       
    dwIntervalMainTask, dwIntervalSecTask      :    DWORD;
    sNameMainTask, sNameSecTask                :    STRING;
    hCurrentTask		                       :    CmpIecTask.RTS_IEC_HANDLE;
    iecResult                                  :    CmpIecTask.RTS_IEC_RESULT;
    sAppName                                   :    STRING := 'Application';
    pIecInfo                                   :    POINTER TO CmpIecTask.Task_Info2;
END_VAR
hCurrentTask := CmpIecTask.IecTaskGetCurrent(pResult := ADR(iecResult));
getCurrentTaskCycleTime:= 0;
IF ((hCurrentTask <> CmpIecTask.RTS_INVALID_HANDLE) AND (iecResult = CmpErrors.Errors.ERR_OK)) THEN
    pIecInfo := CmpIecTask.IecTaskGetInfo3(hIecTask := hCurrentTask, pResult := ADR(iecResult));
    dwIntervalMainTask := pIecInfo^.dwInterval;
    dwCycleTimeMainTask := pIecInfo^.dwCycleTime;
    sNameMainTask := pIecInfo^.pszName^;
	getCurrentTaskCycleTime:= pIecInfo^.dwInterval;
END_IF
END_METHOD

METHOD decrementUINTTimer
VAR_IN_OUT
	input: UINT;
END_VAR
VAR
	step: UINT;
END_VAR
step:= DWORD_TO_UINT(Utils.getCurrentTaskCycleTime() / 1000);
IF(step > input) THEN 
	input:= 0;
ELSE
	input:= input - step;
END_IF
END_METHOD

END_PROGRAM

// Device/Application/Program logic/TypeApplication/ETSDN_Test_PRG
PROGRAM ETSDN_Test_PRG
VAR
	iStepPN: INT:= -1;
	uiTimerIN1TestMs: UINT;
	uiTimerIN2TestMs: UINT;
	uiTimerIP1TestMs: UINT;
	uiTimerIP2TestMs: UINT;
	
	xStepDownAI5V: BOOL;
	iLoopCountAI5V: INT;
	
	xStartIP3: BOOL; 
	wIP3TestOutput: WORD;
	uiTimerIP3TestMs: UINT;
	xStepDownIP3: BOOL;
	iLoopCountIP3: INT;
	
	uiStartTimerButtonPressMs: UINT;
	uiTestDurationTimer: UINT;
	uiTestFailTimerMs: UINT;
	uiTestFailTime: UINT;
	iTestStep: INT:= -1;
	xFailTimerFailValue: BOOL;
	
	wAI5VTestOutput: WORD;
	wIP310VTestOutput: WORD;
	uiTimerAI5VTestMs: UINT;
	
	uiTimerAccTestMs: UINT;
	
	xIP3TestResult, xAITestResult: BOOL;
	xAccZTestResult, xAccYTestResult, xAccXTestResult: BOOL;
	xFirstRLTest: BOOL;
	xAnyRLTestResult, xRL1TestResult, xRL2TestResult, xRL3TestResult: BOOL;
	xIP1TestResult, xIP2TestResult, xIN1TestResult, xIN2TestResult: BOOL;
	
	rPowerSupplyVoltageVolts: REAL;
	wdRLTestTheoricCurrentMilliAmps: DWORD;
	dwRLTestMinCurrent: DWORD;
	dwRLTestMaxCurrent: DWORD;
	
	uiPowerTestFailTimer: UINT;
	ui5VTestFailTimer: UINT;
	uiCANTestFailTimer: UINT;
	TimerAnalog5V: UINT; 
	TimerAnalog10V: UINT;
	Up10V : BOOL; 
	Up5V: BOOL;
	Down: BOOL; 
	
END_VAR

VAR CONSTANT
	RL_TEST_DURATION: UINT:= 500;
	DI_TEST_DURATION: UINT:= 500;
	AI_TEST_DURATION: UINT:= 1500;
	ACC_TEST_TIMEOUT: UINT:= 10000;
	TEST_END_TIMEOUT: UINT:= 20000;
	rAccTolerance: REAL:= 0.3;
	AI_TEST_STEP_TIME: UINT:= 500;
	AI_TEST_STEP_MILLIVOLTS: UINT:= 2000;
	AT_TEST_TOLERANCE_MILLIVOLTS: UINT:= 500;
	RL_TEST_LOAD_OHM: DWORD:= 10;
	RL_TEST_CURRENT_TOLERANCE_PERCENT: DWORD:= 20;
END_VAR

	sysIO.digitalOutput.etsRele_p183.bValue:= EtsdnVar.xPwrSupplyRL1; 
	sysIO.digitalOutput.etsRele_p186.bValue:= EtsdnVar.xPwrSupplyRL2;
	sysIO.digitalOutput.etsRele_p180.bValue:= EtsdnVar.xPwrSupplyRL3;

	
	
	sysIO.digitalOutput.etsIP1_p188.bValue:= EtsdnVar.xPwrSupplyIP1;
	sysIO.digitalOutput.etsIP2_p164.bValue:= EtsdnVar.xPwrSupplyIP2;
	sysIO.digitalOutput.etsIN1_p251.bValue:= EtsdnVar.xPwrSupplyIN1;
	sysIO.digitalOutput.etsIN2_p238.bValue:= EtsdnVar.xPwrSupplyIN2; 
	
	sysIO.digitalOutput.etsPower_p177.bValue:= TRUE;
	
	//________________________________ETSONE________________________________
	sysIO.digitalOutput.etsOnePower_p153.bValue:= TRUE;
	
	sysIO.digitalOutput.etsoneRele_p156.bValue:= EtsOneVar.xOneRL1;
	sysIO.digitalOutput.etsoneRele_p159.bValue:= EtsOneVar.xOneRL2;
	sysIO.digitalOutput.etsIP1_p188.bValue:= EtsOneVar.xOneIP1;
	sysIO.digitalOutput.etsIP2_p164.bValue:= EtsOneVar.xOneIP2;
	sysIO.digitalOutput.etsoneIP3_p194.bValue:= EtsOneVar.xOneIP3;
	
	EtsOneVar.rPwrSupplyOneRL1 := sysIO.digitalOutput.etsoneRele_p156.wCurrent; 
	EtsOneVar.rPwrSupplyOneRL2 := sysIO.digitalOutput.etsoneRele_p159.wCurrent;
	
	
	
	
	IF EtsdnVar.xCycle10V OR EtsOneVar.xCycleOneIP4 THEN 		
		utils.decrementUINT(TimerAnalog10V,1);
			IF TimerAnalog10V = 0 THEN 
				TimerAnalog10V := 2000;
				IF sysIO.voltageOutput.etsAI10V_p185.wOutputVoltageMv = 0 THEN 
					Up10V := TRUE; 
				END_IF
				 
				IF sysIO.voltageOutput.etsAI10V_p185.wOutputVoltageMv > 10000 THEN 
					Up10V := FALSE; 
				END_IF
					
					IF Up10V = TRUE THEN 
						sysIO.voltageOutput.etsAI10V_p185.wOutputVoltageMv := sysIO.voltageOutput.etsAI10V_p185.wOutputVoltageMv +1000;
						ELSE
						sysIO.voltageOutput.etsAI10V_p185.wOutputVoltageMv := sysIO.voltageOutput.etsAI10V_p185.wOutputVoltageMv-1000;			
					END_IF
			END_IF 
	END_IF 	
	
	IF EtsdnVar.xCycle5V THEN 		
		utils.decrementUINT(TimerAnalog5V,1);
			IF TimerAnalog5V = 0 THEN 
				TimerAnalog5V := 2000;
				
				IF sysIO.voltageOutput.etsAI5V_p161.wOutputVoltageMv = 0 THEN 
					Up5V := TRUE;  
				END_IF 
				IF sysIO.voltageOutput.etsAI5V_p161.wOutputVoltageMv > 5000 THEN 
					Up5V := FALSE; 
				END_IF
					
					IF Up5V = TRUE THEN 
						sysIO.voltageOutput.etsAI5V_p161.wOutputVoltageMv := sysIO.voltageOutput.etsAI5V_p161.wOutputVoltageMv +1000;
					ELSE 
						sysIO.voltageOutput.etsAI5V_p161.wOutputVoltageMv := sysIO.voltageOutput.etsAI5V_p161.wOutputVoltageMv-1000;
					END_IF	
			END_IF 
	END_IF
	

	
	
	
	
	
	
// 	
// 	IF EtsOneVar.xCycleOneIP4 THEN 		
// 	utils.decrementUINT(TimerAnalog5V,1);
// 		IF TimerAnalog5V = 0 THEN 
// 			TimerAnalog5V := 2000;
// 			
// 			IF sysIO.voltageOutput.etsAI5V_p161.wOutputVoltageMv = 0 THEN 
// 				Up5V := TRUE;  
// 			END_IF 
// 			IF sysIO.voltageOutput.etsAI5V_p161.wOutputVoltageMv > 5000 THEN 
// 				Up5V := FALSE; 
// 			END_IF
// 				
// 				IF Up5V = TRUE THEN 
// 					sysIO.voltageOutput.etsAI5V_p161.wOutputVoltageMv := sysIO.voltageOutput.etsAI5V_p161.wOutputVoltageMv +1000;
// 				ELSE 
// 					sysIO.voltageOutput.etsAI5V_p161.wOutputVoltageMv := sysIO.voltageOutput.etsAI5V_p161.wOutputVoltageMv-1000;
// 				END_IF	
// 		END_IF 
// 	END_IF
	 
//		sysIO.analogInput.ecuK15_p207.dwValue
//      sysIO.digitalOutput.etsPower_p153.wCurrent
//		sysIO.analogInput.ets5V_p107.dwValue 
//	    sysIO.digitalOutput.etsRele_p156.wCurrent
//      sysIO.digitalOutput.etsRele_p159.wCurrent 
//		sysIO.digitalOutput.etsRele_p180.wCurrent


//      EtsdnVar.xIP1 --> sysIO.digitalOutput.etsIP1_p188.bValue  
//      EtsdnVar.xIP2 --> sysIO.digitalOutput.etsIP2_p164.bValue 
//      EtsdnVar.xIN1 --> sysIO.digitalOutput.etsIN1_p251.bValue 
//      EtsdnVar.xIN2 --> sysIO.digitalOutput.etsIN2_p238.bValue 
//	
//		OUTPUT
//		sysIO.voltageOutput.etsAI_p185.wOutputVoltageMv
//		sysIO.voltageOutput.etsIP3_p161.wOutputVoltageMv:= wIP310VTestOutput;





//       IF NOT system.xTestRunning THEN
//       	IF display.xStartButton THEN
//       		Utils.decrementUINTTimer(uiStartTimerButtonPressMs);
//       		IF uiStartTimerButtonPressMs = 0 THEN
//       			resetVariablesAndStartTest();
//       		END_IF
//       	ELSE
//       		uiStartTimerButtonPressMs:= 100;
//       	END_IF
//       END_IF
//       
//       
//       
//       IF sysIO.analogInput.ecuK15_p207.bValueFresh THEN
//       	rPowerSupplyVoltageVolts:= DWORD_TO_REAL(sysIO.analogInput.ecuK15_p207.dwValue) / 1000;
//       	wdRLTestTheoricCurrentMilliAmps:= (sysIO.analogInput.ecuK15_p207.dwValue / RL_TEST_LOAD_OHM);
//       	dwRLTestMinCurrent:= wdRLTestTheoricCurrentMilliAmps - ((RL_TEST_CURRENT_TOLERANCE_PERCENT * wdRLTestTheoricCurrentMilliAmps) / 100);
//       	dwRLTestMaxCurrent:= wdRLTestTheoricCurrentMilliAmps + ((RL_TEST_CURRENT_TOLERANCE_PERCENT * wdRLTestTheoricCurrentMilliAmps) / 100);
//       END_IF
//       
//       
//       IF system.xTestRunning THEN
//       	// TEST ALIMENTAZIONE continuo
//       	
//       	
//       	IF (sysIO.digitalOutput.etsPower_p153.wCurrent < 50 OR sysIO.digitalOutput.etsPower_p153.wCurrent > 600) OR
//       		(EtsdnVar.rSupplyVoltage < rPowerSupplyVoltageVolts-1 OR EtsdnVar.rSupplyVoltage > rPowerSupplyVoltageVolts+1) THEN
//       		// errore
//       		Utils.decrementUINTTimer(uiPowerTestFailTimer);
//       		IF uiPowerTestFailTimer = 0 THEN system.xPowerTestResult:= FALSE; END_IF
//       	ELSE
//       		uiPowerTestFailTimer:= 500;
//       	END_IF
//       	
//       	
//       	IF sysIO.analogInput.ets5V_p107.dwValue < 4750 OR sysIO.analogInput.ets5V_p107.dwValue > 5200 THEN 
//       		Utils.decrementUINTTimer(ui5VTestFailTimer);
//       		IF ui5VTestFailTimer = 0 THEN system.x5VOutTestResult:= FALSE; END_IF
//       	ELSE
//       		ui5VTestFailTimer:= 500;
//       	END_IF
//       	
//       	IF NOT EtsdnVar.xOnline THEN
//       		Utils.decrementUINTTimer(uiCANTestFailTimer);
//       		IF uiCANTestFailTimer = 0 THEN system.xCanTestResult:= FALSE; END_IF
//       	ELSE
//       		uiCANTestFailTimer:= 1000;
//       	END_IF
//       	
//       END_IF
//       
//       
//       CASE iTestStep OF
//       	-1:
//       		setTestDuration(RL_TEST_DURATION);
//       	
//       	0:
//       		//TEST RELE INIT
//       		sysIO.digitalOutput.etsRele_p156.bValue:= TRUE; 
//       		sysIO.digitalOutput.etsRele_p159.bValue:= TRUE;
//       		sysIO.digitalOutput.etsRele_p180.bValue:= TRUE;
//       		
//       		IF isRLCurrentFresh() AND (
//       			sysIO.digitalOutput.etsRele_p156.wCurrent > 100 OR 
//       			sysIO.digitalOutput.etsRele_p159.wCurrent > 100 OR sysIO.digitalOutput.etsRele_p180.wCurrent > 100
//       		) THEN 
//       			IF NOT mngFailTimer() THEN xAnyRLTestResult:= FALSE; END_IF
//       		END_IF
//       		
//       		IF uiTestDurationTimer = 0 THEN 
//       			setTestDuration(RL_TEST_DURATION);
//       			iTestStep:= iTestStep+1; 
//       		END_IF
//       		
//       	1: 
//       		//TEST RELE 1
//       		EtsdnVar.xRL1:= TRUE;
//       		EtsdnVar.xRL2:= FALSE;
//       		EtsdnVar.xRL3:= FALSE;
//       		IF isRLCurrentFresh() AND (
//       			(sysIO.digitalOutput.etsRele_p156.wCurrent < dwRLTestMinCurrent OR sysIO.digitalOutput.etsRele_p156.wCurrent > dwRLTestMaxCurrent) OR 
//       			sysIO.digitalOutput.etsRele_p159.wCurrent > 10 OR sysIO.digitalOutput.etsRele_p180.wCurrent > 10
//       		) THEN 
//       			IF NOT mngFailTimer() THEN xRL1TestResult:= FALSE; END_IF
//       		END_IF
//       		
//       		IF uiTestDurationTimer = 0 THEN 
//       			setTestDuration(RL_TEST_DURATION);
//       			iTestStep:= iTestStep+1; 
//       		END_IF
//       		
//       	2:
//       		//TEST RELE 2
//       		EtsdnVar.xRL1:= FALSE;
//       		EtsdnVar.xRL2:= TRUE;
//       		EtsdnVar.xRL3:= FALSE;
//       		IF isRLCurrentFresh() AND (
//       			(sysIO.digitalOutput.etsRele_p159.wCurrent < dwRLTestMinCurrent OR sysIO.digitalOutput.etsRele_p159.wCurrent > dwRLTestMaxCurrent) OR 
//       			sysIO.digitalOutput.etsRele_p156.wCurrent > 10 OR sysIO.digitalOutput.etsRele_p180.wCurrent > 10 
//       		) THEN 
//       			IF NOT mngFailTimer() THEN xRL2TestResult:= FALSE; END_IF
//       		END_IF
//       		
//       		IF uiTestDurationTimer = 0 THEN 
//       			setTestDuration(RL_TEST_DURATION);
//       			iTestStep:= iTestStep+1; 
//       		END_IF
//       		
//       	3:
//       		//TEST RELE 3
//       		EtsdnVar.xRL1:= FALSE;
//       		EtsdnVar.xRL2:= FALSE;
//       		EtsdnVar.xRL3:= TRUE;
//       		IF isRLCurrentFresh() AND (
//       			(sysIO.digitalOutput.etsRele_p180.wCurrent < dwRLTestMinCurrent OR sysIO.digitalOutput.etsRele_p180.wCurrent > dwRLTestMaxCurrent) OR 
//       			sysIO.digitalOutput.etsRele_p156.wCurrent > 10 OR sysIO.digitalOutput.etsRele_p159.wCurrent > 10 
//       		) THEN 
//       			IF NOT mngFailTimer() THEN xRL3TestResult:= FALSE; END_IF
//       		END_IF
//       		
//       		IF uiTestDurationTimer = 0 THEN 
//       			EtsdnVar.xRL1:= FALSE;
//       			EtsdnVar.xRL2:= FALSE;
//       			EtsdnVar.xRL3:= FALSE;
//       // 			IF xFirstRLTest THEN
//       // 				xFirstRLTest:= FALSE;
//       // 				setTestDuration(RL_TEST_DURATION);
//       // 				iTestStep:= 0;
//       // 			ELSE
//       				setTestDuration(DI_TEST_DURATION);
//       				iTestStep:= iTestStep+1; 
//       // 			END_IF
//       		END_IF
//       		
//       		
//       	4:
//       		//TEST IP 1
//       		sysIO.digitalOutput.etsIP1_p188.bValue:= TRUE;
//       		IF EtsdnVar.xIP1 <> sysIO.digitalOutput.etsIP1_p188.bValue OR 
//       			EtsdnVar.xIP2 <> sysIO.digitalOutput.etsIP2_p164.bValue OR
//       			EtsdnVar.xIN1 <> sysIO.digitalOutput.etsIN1_p251.bValue OR
//       			EtsdnVar.xIN2 <> sysIO.digitalOutput.etsIN2_p238.bValue THEN
//       			xIP1TestResult:= mngFailTimer();
//       		END_IF
//       		
//       		IF uiTestDurationTimer = 0 THEN 
//       			sysIO.digitalOutput.etsIP1_p188.bValue:= FALSE;
//       			setTestDuration(DI_TEST_DURATION);
//       			iTestStep:= iTestStep+1; 
//       		END_IF
//       		
//       	5:
//       		//TEST IP 2
//       		sysIO.digitalOutput.etsIP2_p164.bValue:= TRUE;
//       		IF EtsdnVar.xIP1 <> sysIO.digitalOutput.etsIP1_p188.bValue OR 
//       			EtsdnVar.xIP2 <> sysIO.digitalOutput.etsIP2_p164.bValue OR
//       			EtsdnVar.xIN1 <> sysIO.digitalOutput.etsIN1_p251.bValue OR
//       			EtsdnVar.xIN2 <> sysIO.digitalOutput.etsIN2_p238.bValue THEN
//       			xIP2TestResult:= mngFailTimer();
//       		END_IF
//       		
//       		IF uiTestDurationTimer = 0 THEN 
//       			sysIO.digitalOutput.etsIP2_p164.bValue:= FALSE;
//       			setTestDuration(DI_TEST_DURATION);
//       			iTestStep:= iTestStep+1; 
//       		END_IF
//       		
//       	6:
//       		//TEST IN 1
//       		sysIO.digitalOutput.etsIN1_p251.bValue:= TRUE;
//       		IF EtsdnVar.xIP1 <> sysIO.digitalOutput.etsIP1_p188.bValue OR 
//       			EtsdnVar.xIP2 <> sysIO.digitalOutput.etsIP2_p164.bValue OR
//       			EtsdnVar.xIN1 <> sysIO.digitalOutput.etsIN1_p251.bValue OR
//       			EtsdnVar.xIN2 <> sysIO.digitalOutput.etsIN2_p238.bValue THEN
//       			xIN1TestResult:= mngFailTimer();
//       		END_IF
//       		
//       		IF uiTestDurationTimer = 0 THEN 
//       			sysIO.digitalOutput.etsIN1_p251.bValue:= FALSE;
//       			setTestDuration(DI_TEST_DURATION);
//       			iTestStep:= iTestStep+1; 
//       		END_IF
//       		
//       	7:
//       		//TEST IN 2
//       		sysIO.digitalOutput.etsIN2_p238.bValue:= TRUE;
//       		IF EtsdnVar.xIP1 <> sysIO.digitalOutput.etsIP1_p188.bValue OR 
//       			EtsdnVar.xIP2 <> sysIO.digitalOutput.etsIP2_p164.bValue OR
//       			EtsdnVar.xIN1 <> sysIO.digitalOutput.etsIN1_p251.bValue OR
//       			EtsdnVar.xIN2 <> sysIO.digitalOutput.etsIN2_p238.bValue THEN
//       			xIN2TestResult:= mngFailTimer();
//       		END_IF
//       		
//       		IF uiTestDurationTimer = 0 THEN 
//       			sysIO.digitalOutput.etsIN2_p238.bValue:= FALSE;
//       			setTestDuration(AI_TEST_DURATION);
//       			iTestStep:= iTestStep+1; 
//       		END_IF
//       		
//       	8:
//       		// TEST AI 0-5V
//       		IF uiTimerAI5VTestMs = 0 THEN
//       			// step aumento tensione
//       			uiTimerAI5VTestMs:= AI_TEST_STEP_TIME;
//       			
//       			IF wAI5VTestOutput >= 5000 THEN
//       				xStepDownAI5V:= TRUE;
//       				iLoopCountAI5V:= iLoopCountAI5V + 1;
//       			ELSIF wAI5VTestOutput = 0 THEN
//       				xStepDownAI5V:= FALSE;
//       			END_IF
//       			
//       			IF xStepDownAI5V THEN
//       				wAI5VTestOutput:= wAI5VTestOutput - AI_TEST_STEP_MILLIVOLTS;
//       			ELSE
//       				wAI5VTestOutput:= wAI5VTestOutput + AI_TEST_STEP_MILLIVOLTS;
//       			END_IF
//       			IF wAI5VTestOutput > 5000 THEN wAI5VTestOutput:= 5000; END_IF
//       			sysIO.voltageOutput.etsAI_p185.wOutputVoltageMv:= wAI5VTestOutput;
//       		END_IF
//       		
//       		IF (EtsdnVar.rAI * 1000) < (wAI5VTestOutput -AT_TEST_TOLERANCE_MILLIVOLTS) OR (EtsdnVar.rAI * 1000) > (wAI5VTestOutput +AT_TEST_TOLERANCE_MILLIVOLTS)  THEN
//       			xAITestResult:= mngFailTimer();
//       		END_IF
//       		
//       		Utils.decrementUINTTimer(uiTimerAI5VTestMs);
//       		
//       		IF uiTestDurationTimer = 0 THEN 
//       			setTestDuration(AI_TEST_DURATION);
//       			iTestStep:= iTestStep+1; 
//       		END_IF
//       		
//       	9:
//       		// TEST IP3 0-10V
//       		IF uiTimerAI5VTestMs = 0 THEN
//       			// step aumento tensione
//       			uiTimerAI5VTestMs:= AI_TEST_STEP_TIME;
//       			
//       			IF wIP310VTestOutput >= 10000 THEN
//       				xStepDownAI5V:= TRUE;
//       				iLoopCountAI5V:= iLoopCountAI5V + 1;
//       			ELSIF wIP310VTestOutput = 0 THEN
//       				xStepDownAI5V:= FALSE;
//       			END_IF
//       			
//       			IF xStepDownAI5V THEN
//       				wIP310VTestOutput:= wIP310VTestOutput - AI_TEST_STEP_MILLIVOLTS*2;
//       			ELSE
//       				wIP310VTestOutput:= wIP310VTestOutput + AI_TEST_STEP_MILLIVOLTS*2;
//       			END_IF
//       			IF wIP310VTestOutput > 10000 THEN wIP310VTestOutput:= 5000; END_IF
//       			sysIO.voltageOutput.etsIP3_p161.wOutputVoltageMv:= wIP310VTestOutput;
//       		END_IF
//       		
//       		IF (EtsdnVar.rIP3 * 1000) < (wIP310VTestOutput -AT_TEST_TOLERANCE_MILLIVOLTS) OR (EtsdnVar.rIP3 * 1000) > (wIP310VTestOutput +AT_TEST_TOLERANCE_MILLIVOLTS) THEN
//       			xIP3TestResult:= mngFailTimer();
//       		END_IF
//       		
//       		Utils.decrementUINTTimer(uiTimerAI5VTestMs);
//       		
//       		IF uiTestDurationTimer = 0 THEN 
//       			setTestDuration(ACC_TEST_TIMEOUT);
//       			iTestStep:= iTestStep+1; 
//       		END_IF
//       		
//       	10: // accelerometro Z
//       		system.iAccTestStep:= 0;
//       		IF (EtsdnVar.rZ > 1-rAccTolerance AND EtsdnVar.rZ < 1+rAccTolerance) AND (EtsdnVar.rY > -rAccTolerance AND EtsdnVar.rY < rAccTolerance) AND (EtsdnVar.rX > -rAccTolerance AND EtsdnVar.rX < rAccTolerance) THEN
//       			// posizione OK
//       			uiTimerAccTestMs:= uiTimerAccTestMs+10;
//       			IF uiTimerAccTestMs > 500 THEN
//       				xAccZTestResult:= TRUE; 
//       				uiTimerAccTestMs:= 0;
//       				iTestStep:= iTestStep+1; 
//       			END_IF
//       		END_IF
//       		
//       		IF uiTestDurationTimer = 0 THEN 
//       			setTestDuration(ACC_TEST_TIMEOUT);
//       			iTestStep:= iTestStep+1; 
//       		END_IF
//       		
//       	11: // accelerometro Y
//       		system.iAccTestStep:= 1;
//       		IF (EtsdnVar.rY > -1-rAccTolerance AND EtsdnVar.rY < -1+rAccTolerance) AND (EtsdnVar.rZ > -rAccTolerance AND EtsdnVar.rZ < rAccTolerance) AND (EtsdnVar.rX > -rAccTolerance AND EtsdnVar.rX < rAccTolerance) THEN
//       			// posizione OK
//       			uiTimerAccTestMs:= uiTimerAccTestMs+10;
//       			IF uiTimerAccTestMs > 500 THEN
//       				xAccYTestResult:= TRUE; 
//       				uiTimerAccTestMs:= 0;
//       				iTestStep:= iTestStep+1; 
//       			END_IF
//       		END_IF
//       		
//       		IF uiTestDurationTimer = 0 THEN 
//       // 			setTestDuration(ACC_TEST_TIMEOUT);
//       			setTestDuration(TEST_END_TIMEOUT);
//       			iTestStep:= iTestStep+1; 
//       		END_IF
//       		
//       	12: // accelerometro X skip chiesto da Andrea
//       		iTestStep:= iTestStep+1; 
//       		xAccXTestResult:= TRUE; 
//       // 		system.iAccTestStep:= 2;
//       // 		IF (etsdn.rX > 1-rAccTolerance AND etsdn.rX < 1+rAccTolerance) AND (etsdn.rY > -rAccTolerance AND etsdn.rY < rAccTolerance) AND (etsdn.rZ > -rAccTolerance AND etsdn.rZ < rAccTolerance) THEN
//       // 			// posizione OK
//       // 			uiTimerAccTestMs:= uiTimerAccTestMs+10;
//       // 			IF uiTimerAccTestMs > 500 THEN
//       // 				xAccXTestResult:= TRUE; 
//       // 				uiTimerAccTestMs:= 0;
//       // 				iTestStep:= iTestStep+1; 
//       // 			END_IF
//       // 		END_IF
//       // 		
//       // 		IF uiTestDurationTimer = 0 THEN 
//       // 			setTestDuration(TEST_END_TIMEOUT);
//       // 			iTestStep:= iTestStep+1; 
//       // 		END_IF
//       		
//       	13:
//       		endTest();
//       		setTestDuration(RL_TEST_DURATION);
//       		IF uiTestDurationTimer = 0 THEN
//       			iTestStep:= -1; 
//       		END_IF
//       		
//       	
//       END_CASE
//       
//       system.xAnalogInTestResult:= xIP3TestResult AND xAITestResult;
//       system.xAccelerometerTestResult:= xAccZTestResult AND xAccYTestResult AND xAccXTestResult;
//       system.xReleTestResult:= xAnyRLTestResult AND xRL1TestResult AND xRL2TestResult AND xRL3TestResult;
//       system.xDigitalInTestResult:= xIP1TestResult AND xIP2TestResult AND xIN1TestResult AND xIN2TestResult;
//       IF iTestStep >= 0 THEN system.byTestPercentage:= REAL_TO_BYTE((INT_TO_REAL(iTestStep)*100)/13); END_IF
//       Utils.decrementUINTTimer(uiTestDurationTimer);

METHOD PRIVATE endTest
VAR_INPUT
END_VAR
system.xTestResult:= (
	system.xCanTestResult AND
	system.xDigitalInTestResult AND
	system.xAnalogInTestResult AND
	system.xPowerTestResult AND
	system.x5VOutTestResult AND
	system.xAccelerometerTestResult AND
	system.xReleTestResult
);
system.xTestRunning:= FALSE;
system.xTestResultValid:= TRUE;

EtsdnVar.xRL1:= FALSE;
EtsdnVar.xRL2:= FALSE;
EtsdnVar.xRL3:= FALSE;

sysIO.digitalOutput.etsonePower_p153.bValue:= FALSE;
sysIO.digitalOutput.etsRele_p183.bValue:= FALSE; 
sysIO.digitalOutput.etsRele_p186.bValue:= FALSE;
sysIO.digitalOutput.etsRele_p180.bValue:= FALSE;

sysIO.digitalOutput.etsIP1_p188.bValue:= FALSE;
sysIO.digitalOutput.etsIP2_p164.bValue:= FALSE;
sysIO.digitalOutput.etsIN1_p251.bValue:= FALSE;
sysIO.digitalOutput.etsIN2_p238.bValue:= FALSE;

sysIO.voltageOutput.etsAI10V_p185.wOutputVoltageMv:= 0;
sysIO.voltageOutput.etsAI5V_p161.wOutputVoltageMv:= 0;
END_METHOD

METHOD PRIVATE setTestDuration
VAR_INPUT
	uiDurationMs: UINT;
END_VAR
uiTestDurationTimer:= uiDurationMs;
uiTestFailTime:= uiTestDurationTimer / 2;
uiTestFailTimerMs:= 0;
xFailTimerFailValue:= TRUE;
END_METHOD

METHOD PRIVATE resetVariablesAndStartTest
VAR_INPUT
END_VAR
system.xTestResult:= FALSE;
system.xTestResultValid:= FALSE;

system.xCanTestResult:= TRUE;
system.xDigitalInTestResult:= TRUE;
system.xAnalogInTestResult:= TRUE;
system.xPowerTestResult:= TRUE;
system.x5VOutTestResult:= TRUE;
system.xAccelerometerTestResult:= TRUE;
system.xReleTestResult:= TRUE;
xIP3TestResult:= TRUE;
xAITestResult:= TRUE;
xAccZTestResult:= FALSE;
xAccYTestResult:= FALSE;
xAccXTestResult:= FALSE;
xFirstRLTest:= TRUE;
xAnyRLTestResult:= TRUE;
xRL1TestResult:= TRUE;
xRL2TestResult:= TRUE;
xRL3TestResult:= TRUE;

system.iAccTestStep:= -1;

system.xTestRunning:= TRUE;
system.byTestPercentage:= 0;

iTestStep:= 0;
wAI5VTestOutput:= 0;
wIP310VTestOutput:= 0;

uiPowerTestFailTimer:= 2000;
ui5VTestFailTimer:= 2000;
uiCANTestFailTimer:= 2000;
	
sysIO.digitalOutput.etsonePower_p153.bValue:= TRUE;
END_METHOD

METHOD PRIVATE mngFailTimer: BOOL;
VAR_INPUT
END_VAR
uiTestFailTimerMs:= uiTestFailTimerMs + DWORD_TO_UINT(Utils.getCurrentTaskCycleTime() / 1000);
IF uiTestFailTimerMs >= uiTestFailTime THEN
	xFailTimerFailValue:= FALSE;
END_IF
mngFailTimer:= xFailTimerFailValue;
END_METHOD

METHOD PRIVATE isRLCurrentFresh : BOOL	
VAR_INPUT
END_VAR
isRLCurrentFresh:= 
	sysIO.digitalOutput.etsRele_p183.bCurrentFresh AND
	sysIO.digitalOutput.etsRele_p186.bCurrentFresh AND
	sysIO.digitalOutput.etsRele_p180.bCurrentFresh;
END_METHOD

END_PROGRAM

// Device/Application/Program logic/Tasks/MAIN
PROGRAM MAIN
VAR
	xStop: BOOL:= FALSE;
	init : BOOL := FALSE;
	INIT_STEP : UINT:=0;
	result : RTS_IEC_RESULT;
	DeviceName : WSTRING(255) := "";
	DeviceNameLen : UDINT := 255;
	TargetId : DWORD := 0;
	NodeName : WSTRING(255) := "";
	NodeNameLen : UDINT := 255;
	OperatingSystemId : UDINT := 0;
	ProcessorId : UDINT := 0;
	SerialNumber : POINTER TO STRING := 0;
	SerialNumberLen : DINT := 255;
	TargetType : DWORD := 0;
	VendorName : WSTRING(255) := "";
	VendorNameLen : UDINT := 255;
	Version : DWORD := 0;
	
	error_code : lib500_types.IO_ERRORTYPE := lib500_types.IO_ERRORTYPE.IO_E_OK;
		
	shutdownCounterMillis: UDINT:= 30 * 1000;
	uiPowerOnTimeMs: UINT:= 0;
END_VAR

// check, if in init phase
IF (init = FALSE) THEN
	CASE INIT_STEP OF
	0:	
		// SysTargetGetDeviceName()
		result := SysTarget.SysTargetGetDeviceName(
			pwszName:= ADR(DeviceName),
			pnMaxLength:= ADR(DeviceNameLen));
		
		// SysTargetGetId()
		result := SysTarget.SysTargetGetId(
			pulTargetId:= ADR(TargetId));
		
		// SysTargetGetNodeName()
		result := SysTarget.SysTargetGetNodeName(
			pwszName:= ADR(NodeName), 
			pnMaxLength:= ADR(NodeNameLen));
		
		// SysTargetGetOperatingSystemId()
		result := SysTarget.SysTargetGetOperatingSystemId(
			pudiOperatingSystemId:= ADR(OperatingSystemId));
		
		// SysTargetGetProcessorId()
		result := SysTarget.SysTargetGetProcessorId(
			pudiProcessorId:= ADR(ProcessorId));
		
		// SysTargetGetSerialNumber()
		result := SysTarget.SysTargetGetSerialNumber(
			ppsSerialNumber:= ADR(SerialNumber),
			pnMaxLen:= ADR(SerialNumberLen));
		
		// SysTargetGetType()
		result := SysTarget.SysTargetGetType(
			pulType:= ADR(TargetType));
		
		// SysTargetGetVendorName()
		result := SysTarget.SysTargetGetVendorName(
			pwszName:= ADR(VendorName),
			pnMaxLength:= ADR(VendorNameLen));
		
		// SysTargetGetVersion()
		result := SysTarget.SysTargetGetVersion(
			pulVersion:= ADR(Version));
		
		IF DeviceName = "HY-TTC 540" THEN
			GVL.MODELLO_CENTRALINA:= 1;
		ELSIF DeviceName = "HY-TTC 580" THEN
			GVL.MODELLO_CENTRALINA:= 2;
		END_IF								 
		 
		INIT_STEP:=INIT_STEP+1;	
	1:	
		//MNG_RW_EEPROM();
		//IF EEPROM.EEPROM_ST = TRUE THEN
			checkParameters();
			INIT_STEP:=INIT_STEP+1;	
		//END_IF
		
	2:
		IF NOT sysIO.bIOInitialized THEN
			initializeIO();
			IF sysIO.bIOInitialized THEN INIT_STEP:=INIT_STEP+1; END_IF
		END_IF
		
	3:		
		IF NOT fieldbus.bCanbusInitialized THEN
			setupCanbus();
		ELSE
// 			J1939_PRG.canbus:= fieldbus.can[1];	
// 			J1939.xRedirectMessages:= TRUE;
// 			J1939.xSendPGNRequest:= TRUE;
			init:= TRUE;
		END_IF
	END_CASE							  
END_IF

IF (init = TRUE) THEN	
	IF xStop THEN RETURN; END_IF
	checkParameters();
	
	io_module.getInputs();	
	IO.xECUK15:= sysIO.analogInput.ecuK15_p207.dwValue > 10000; 
	
	IF (IO.xECUK15) THEN
		// Esecuzione regolare
		mainLoop();
	ELSIF NOT GVL.xAllowSystemShutdown THEN
		postrun();
	ELSE
		shutdown();
	END_IF
	
	IF uiPowerOnTimeMs < 65000 THEN uiPowerOnTimeMs:= uiPowerOnTimeMs +10; END_IF
	
	UI_PRG();
	io_module.setOutputs();
	system.xFirstCycle:= FALSE;
	
END_IF

METHOD PRIVATE mainLoop
VAR_INPUT
END_VAR
//mngCanbusStatus();	
//J1939_PRG();

ETSDN_Test_PRG();

IF system.xHazardStatus THEN
	shutdownCounterMillis:= 6 * 60 * 60 * 1000; // 6 ore
ELSE
	shutdownCounterMillis:= 30 * 1000;
END_IF
END_METHOD

ACTION postrun:
Utils.decrementUDINT(shutdownCounterMillis, 10);
GVL.xAllowSystemShutdown:= ((NOT system.xHazardStatus) OR 
							(shutdownCounterMillis = 0)) AND
							uiPowerOnTimeMs > 10000; // devono essere passati almeno 10 secondi dal key-on per poter spegnere (per K15 display)
END_ACTION

ACTION shutdown:

error_code:= lib500.IO_POWER_Set(lib500_types.IO_POWER_CHANNEL.IO_K15, lib500_types.IO_POWER_STATE.IO_POWER_OFF);
END_ACTION

METHOD PRIVATE checkParameters
VAR_INPUT
END_VAR
END_METHOD

ACTION setupCanbus:
IF NOT fieldbus.bCanbusInitialized THEN
	fieldbus.can[0].bActive:= FALSE;
	fieldbus.can[1].bActive:= TRUE; 
	fieldbus.can[2].bActive:= true; 
	fieldbus.can[3].bActive:= TRUE;
	fieldbus.can[4].bActive:= TRUE; 
	fieldbus.can[5].bActive:= FALSE;
	fieldbus.can[6].bActive:= FALSE;
	fieldbus.bCanbusInitialized:= initializeCanbus();	
END_IF
END_ACTION

END_PROGRAM

// Device/Application/Modules/IOs/Types/initializeIO
PROGRAM initializeIO
VAR
	bInstantiated: BOOL:= FALSE;
END_VAR

VAR CONSTANT
	TTC_540: BYTE:= 1;
	TTC_580: BYTE:= 2;
END_VAR

IF NOT bInstantiated THEN 
	instantiatePowerStages();
	
	instantiateDigitalInputs();
	instantiateAnalogInputs();
	instantiatePWDInputs();
	
	instantiateDigitalOutputs();
	instantiatePWMOutputs();
	instantiateVoltageOutputs();
	
	bInstantiated:= TRUE;
END_IF

sysIO.bIOInitialized:= io_module.initializeIO(GVL.MODELLO_CENTRALINA);

METHOD PRIVATE instantiateAnalogInputs
VAR_INPUT
END_VAR
io_module.instantiateADC(	
	outPointer:= ADR(sysIO.analogInput.ecuK15_p207), 
	byChannel:= lib500_types.IO_ADC_CHANNEL.IO_ADC_K15, 
	byPullType:= lib500_types.IO_ADC_PUPD.IO_ADC_NO_PULL,
	stADCType:= lib500_types.IO_ADC_TYPE.IO_ADC_ABSOLUTE,
	stADCRange:= lib500_types.IO_ADC_RANGE.IO_ADC_RANGE_32V,
	stADCSensorSupply:= lib500_types.IO_SENSOR_SUPPLY.IO_SENSOR_SUPPLY_0
);

io_module.instantiateADC(
	outPointer:= ADR(sysIO.analogInput.etsone5V_107), 
	byChannel:= lib500_types.IO_ADC_CHANNEL.IO_ADC_08, 
	byPullType:= lib500_types.IO_ADC_PUPD.IO_ADC_NO_PULL,
	stADCType:= lib500_types.IO_ADC_TYPE.IO_ADC_ABSOLUTE,
	stADCRange:= lib500_types.IO_ADC_RANGE.IO_ADC_RANGE_5V,
	stADCSensorSupply:= lib500_types.IO_SENSOR_SUPPLY.IO_PIN_NONE
);

io_module.instantiateADC(
	outPointer:= ADR(sysIO.analogInput.ets5V_p131), 
	byChannel:= lib500_types.IO_ADC_CHANNEL.IO_ADC_09, 
	byPullType:= lib500_types.IO_ADC_PUPD.IO_ADC_NO_PULL,
	stADCType:= lib500_types.IO_ADC_TYPE.IO_ADC_ABSOLUTE,
	stADCRange:= lib500_types.IO_ADC_RANGE.IO_ADC_RANGE_5V,
	stADCSensorSupply:= lib500_types.IO_SENSOR_SUPPLY.IO_PIN_NONE
);
END_METHOD

METHOD PRIVATE instantiatePVGOutputs
VAR_INPUT
END_VAR
//io_module.instantiatePVG(			
//	outPointer:= ADR(sysIO.pvgOutput._p161),
//	byChannel:= lib500_types.IO_PWD_CHANNEL.IO_PWD_04,
//	5000
//);
END_METHOD

 METHOD PRIVATE instantiateDigitalOutputs
VAR_INPUT
END_VAR
io_module.instantiateDO(				
	outPointer:= ADR(sysIO.digitalOutput.etsonePower_p153),
	byChannel:= lib500_types.IO_DO_CHANNEL.IO_DO_16
);

io_module.instantiateDO(				
	outPointer:= ADR(sysIO.digitalOutput.etsPower_p177),
	byChannel:= lib500_types.IO_DO_CHANNEL.IO_DO_17
);

io_module.instantiateDO(				
	outPointer:= ADR(sysIO.digitalOutput.etsIP1_p188),
	byChannel:= lib500_types.IO_DO_CHANNEL.IO_DO_54
);


io_module.instantiateDO(				
	outPointer:= ADR(sysIO.digitalOutput.etsRele_p186),
	byChannel:= lib500_types.IO_DO_CHANNEL.IO_DO_22
);

io_module.instantiateDO(				
	outPointer:= ADR(sysIO.digitalOutput.etsoneRele_p156),
	byChannel:= lib500_types.IO_DO_CHANNEL.IO_DO_18
);

io_module.instantiateDO(				
	outPointer:= ADR(sysIO.digitalOutput.etsRele_p180),
	byChannel:= lib500_types.IO_DO_CHANNEL.IO_DO_19
);

io_module.instantiateDO(				
	outPointer:= ADR(sysIO.digitalOutput.etsRele_p183),
	byChannel:= lib500_types.IO_DO_CHANNEL.IO_DO_21
);


io_module.instantiateDO(				
	outPointer:= ADR(sysIO.digitalOutput.etsoneRele_p159),
	byChannel:= lib500_types.IO_DO_CHANNEL.IO_DO_20
);
io_module.instantiateDO(				
	outPointer:= ADR(sysIO.digitalOutput.etsIN1_p251),
	byChannel:= lib500_types.IO_DO_CHANNEL.IO_DO_08
);
io_module.instantiateDO(				
	outPointer:= ADR(sysIO.digitalOutput.etsIP2_p164),
	byChannel:= lib500_types.IO_DO_CHANNEL.IO_DO_55
);

io_module.instantiateDO(				
	outPointer:= ADR(sysIO.digitalOutput.etsoneIP3_p194),
	byChannel:= lib500_types.IO_DO_CHANNEL.IO_DO_58
);

io_module.instantiateDO(				
	outPointer:= ADR(sysIO.digitalOutput.etsIN2_p238),
	byChannel:= lib500_types.IO_DO_CHANNEL.IO_DO_09
);
END_METHOD

